REGION Network 69: EM Status Homed
   RUNG wire#powerrail
      Contact( "Unit1.Em4.ControlNodes".mainPnP.preOperationCheck.partNoDetect1 )
      wire#w1
      Contact( "Unit1.Em4.ControlNodes".alignTable.preOperationCheck.partNoDetect1 )
      wire#w2
      Contact( "Unit1.Em4.ControlNodes".ngPnP.preOperationCheck.partNoDetect )
      wire#w3
      I_Contact( #unitStatus.specialFunctions.dryRun )
      wire#w4
      Coil( "Unit1.Em4.ControlNodes".em.status.homed )
      Coil( #emFeedback.status.homed )
   END_RUNG
   RUNG wire#powerrail
      Contact( "Unit1.Em4.ControlNodes".mainPnP.preOperationCheck.partNoDetect2 )
   END_RUNG wire#w1
   RUNG wire#powerrail
      Contact( "Unit1.Em4.ControlNodes".mainPnP.preOperationCheck.partDetect1 )
   END_RUNG wire#w1
   RUNG wire#powerrail
      Contact( "Unit1.Em4.ControlNodes".mainPnP.preOperationCheck.partDetect2 )
   END_RUNG wire#w1
   RUNG wire#powerrail
      Contact( "Unit1.Em4.ControlNodes".mainPnP.preOperationCheck.partNG )
   END_RUNG wire#w1
   RUNG wire#powerrail
      Contact( "Unit1.Em4.ControlNodes".mainPnP.preOperationCheck.PartDetect1_1 )
   END_RUNG wire#w1
   RUNG wire#w1
      Contact( "Unit1.Em4.ControlNodes".alignTable.preOperationCheck.partDetect1 )
   END_RUNG wire#w2
   RUNG wire#w1
      Contact( "Unit1.Em4.ControlNodes".alignTable.preOperationCheck.partDetect2 )
   END_RUNG wire#w2
   RUNG wire#w2
      Contact( "Unit1.Em4.ControlNodes".ngPnP.preOperationCheck.partDetect )
   END_RUNG wire#w3
   RUNG wire#powerrail
      Contact( #unitStatus.specialFunctions.dryRun )
   END_RUNG wire#w4
   // the same network as SCL:
   "Unit1.Em4.ControlNodes".em.status.homed := (("Unit1.Em4.ControlNodes".mainPnP.preOperationCheck.partNoDetect1 OR "Unit1.Em4.ControlNodes".mainPnP.preOperationCheck.partNoDetect2 OR "Unit1.Em4.ControlNodes".mainPnP.preOperationCheck.partDetect1 OR "Unit1.Em4.ControlNodes".mainPnP.preOperationCheck.partDetect2 OR "Unit1.Em4.ControlNodes".mainPnP.preOperationCheck.partNG OR "Unit1.Em4.ControlNodes".mainPnP.preOperationCheck.PartDetect1_1) AND ("Unit1.Em4.ControlNodes".alignTable.preOperationCheck.partNoDetect1 OR "Unit1.Em4.ControlNodes".alignTable.preOperationCheck.partDetect1 OR "Unit1.Em4.ControlNodes".alignTable.preOperationCheck.partDetect2) AND ("Unit1.Em4.ControlNodes".ngPnP.preOperationCheck.partNoDetect OR "Unit1.Em4.ControlNodes".ngPnP.preOperationCheck.partDetect) AND NOT #unitStatus.specialFunctions.dryRun) OR #unitStatus.specialFunctions.dryRun;
   #emFeedback.status.homed := "Unit1.Em4.ControlNodes".em.status.homed;
END_REGION

REGION Network 70: EM Status Motion Ready
   RUNG wire#powerrail
      I_Contact( #instMainPnPHomeJob10.jobStatus.active )
      I_Contact( #instMainPnPLoadJob2.jobStatus.active )
      I_Contact( #instMainPnPUnloadJob3.jobStatus.active )
      I_Contact( #instMainPnPAvoidJob4.jobStatus.active )
      I_Contact( #instMainPnPOneLoadJob5.jobStatus.active )
      I_Contact( #instMainPnPOneUnLoadJob6.jobStatus.active )
      I_Contact( #instMainPnPDownWaitJob7.jobStatus.active )
      Coil( "Unit1.EmNodes".emRelations.em04."Bool"[10] )
   END_RUNG
   // the same network as SCL:
   "Unit1.EmNodes".emRelations.em04."Bool"[10] := NOT #instMainPnPHomeJob10.jobStatus.active AND NOT #instMainPnPLoadJob2.jobStatus.active AND NOT #instMainPnPUnloadJob3.jobStatus.active AND NOT #instMainPnPAvoidJob4.jobStatus.active AND NOT #instMainPnPOneLoadJob5.jobStatus.active AND NOT #instMainPnPOneUnLoadJob6.jobStatus.active AND NOT #instMainPnPDownWaitJob7.jobStatus.active;
END_REGION

REGION Network 72: Call Sequence [Main P&P]
   // Call the sequence. This contains the main logic of the equipment module
   RUNG wire#powerrail
      #InstSequenceMainPnP()
   END_RUNG
   // the same network as SCL:
   #InstSequenceMainPnP();   // "Unit1.Em4.Sequence_1_MainPnP"
END_REGION

REGION Network 73: Call Sequence [Align Table]
   // Call the sequence. This contains the main logic of the equipment module
   RUNG wire#powerrail
      #InstSequenceAlignTable()
   END_RUNG
   // the same network as SCL:
   #InstSequenceAlignTable();   // "Unit1.Em4.Sequence_2_AlignTable"
END_REGION

REGION Network 74: Call Sequence [NG P&P]
   // Call the sequence. This contains the main logic of the equipment module
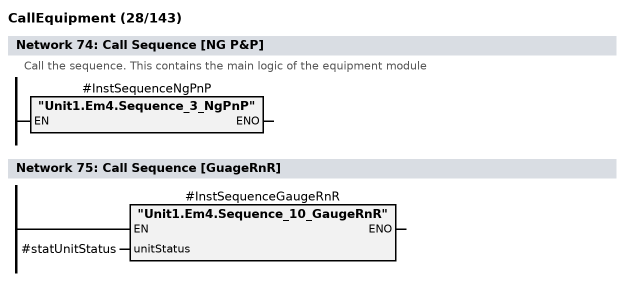
   RUNG wire#powerrail
      #InstSequenceNgPnP()
   END_RUNG
   // the same network as SCL:
   #InstSequenceNgPnP();   // "Unit1.Em4.Sequence_3_NgPnP"
END_REGION

REGION Network 75: Call Sequence [GuageRnR]
   RUNG wire#powerrail
      #InstSequenceGaugeRnR(unitStatus := #statUnitStatus)
   END_RUNG
   // the same network as SCL:
   #InstSequenceGaugeRnR(unitStatus := #statUnitStatus);   // "Unit1.Em4.Sequence_10_GaugeRnR"
END_REGION

REGION Network 76: *************** Control Modules (Axis) *******************
   // Call control modules that are actuators after the em logic (jobs and sequence), so that the latest commands are applied to the actuators.
END_REGION

REGION Network 77: Reset CMS
   // Reset Axis when the unit is in the resetting state.
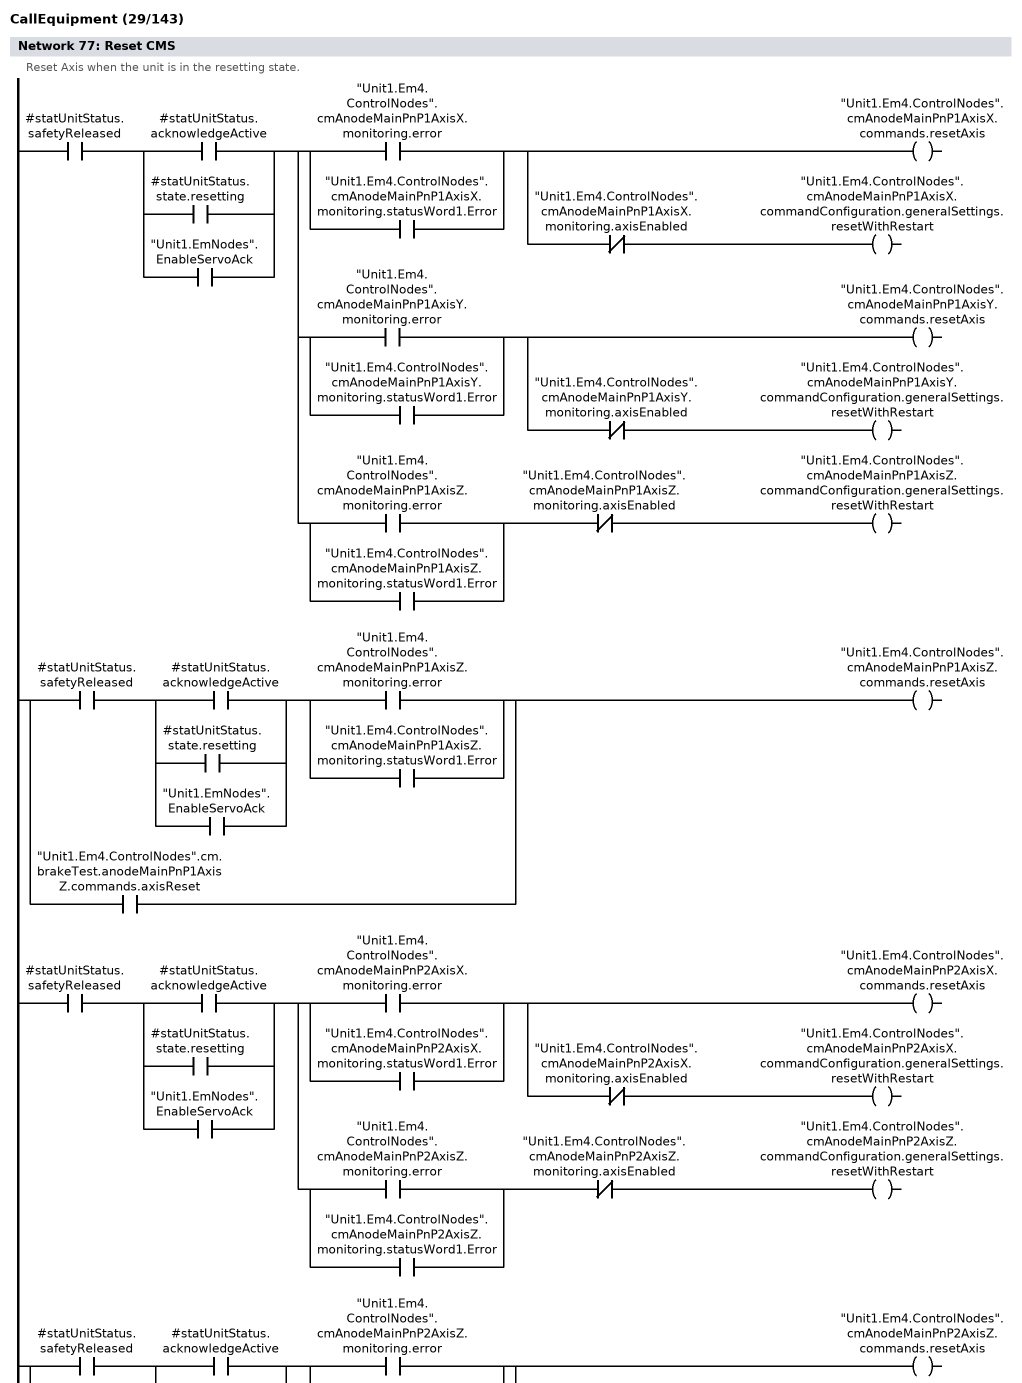
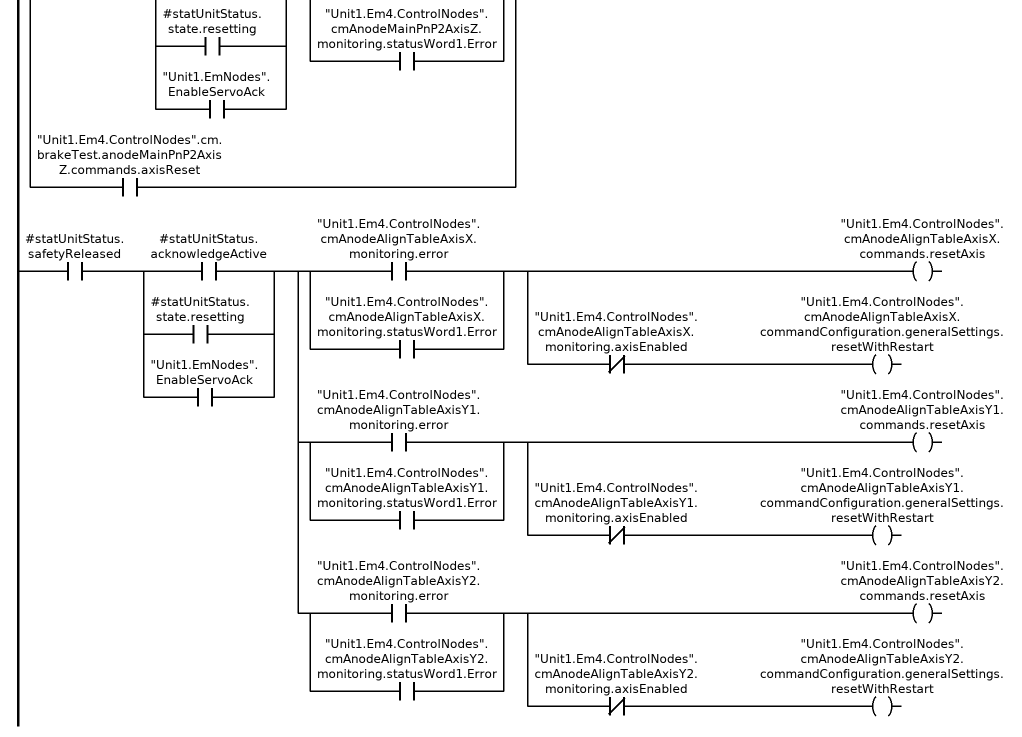
   RUNG wire#powerrail
      Contact( #statUnitStatus.safetyReleased )
      wire#w1
      Contact( #statUnitStatus.acknowledgeActive )
      wire#w2
      Contact( "Unit1.Em4.ControlNodes".cmAnodeMainPnP1AxisX.monitoring.error )
      wire#w3
      Coil( "Unit1.Em4.ControlNodes".cmAnodeMainPnP1AxisX.commands.resetAxis )
   END_RUNG
   RUNG wire#w1
      Contact( #statUnitStatus.state.resetting )
   END_RUNG wire#w2
   RUNG wire#w1
      Contact( "Unit1.EmNodes".EnableServoAck )
   END_RUNG wire#w2
   RUNG wire#w2
      Contact( "Unit1.Em4.ControlNodes".cmAnodeMainPnP1AxisX.monitoring.statusWord1.Error )
   END_RUNG wire#w3
   RUNG wire#w3
      I_Contact( "Unit1.Em4.ControlNodes".cmAnodeMainPnP1AxisX.monitoring.axisEnabled )
      Coil( "Unit1.Em4.ControlNodes".cmAnodeMainPnP1AxisX.commandConfiguration.generalSettings.resetWithRestart )
   END_RUNG
   RUNG wire#w2
      Contact( "Unit1.Em4.ControlNodes".cmAnodeMainPnP1AxisY.monitoring.error )
      wire#w4
      Coil( "Unit1.Em4.ControlNodes".cmAnodeMainPnP1AxisY.commands.resetAxis )
   END_RUNG
   RUNG wire#w2
      Contact( "Unit1.Em4.ControlNodes".cmAnodeMainPnP1AxisY.monitoring.statusWord1.Error )
   END_RUNG wire#w4
   RUNG wire#w4
      I_Contact( "Unit1.Em4.ControlNodes".cmAnodeMainPnP1AxisY.monitoring.axisEnabled )
      Coil( "Unit1.Em4.ControlNodes".cmAnodeMainPnP1AxisY.commandConfiguration.generalSettings.resetWithRestart )
   END_RUNG
   RUNG wire#w2
      Contact( "Unit1.Em4.ControlNodes".cmAnodeMainPnP1AxisZ.monitoring.error )
      wire#w5
      I_Contact( "Unit1.Em4.ControlNodes".cmAnodeMainPnP1AxisZ.monitoring.axisEnabled )
      Coil( "Unit1.Em4.ControlNodes".cmAnodeMainPnP1AxisZ.commandConfiguration.generalSettings.resetWithRestart )
   END_RUNG
   RUNG wire#w2
      Contact( "Unit1.Em4.ControlNodes".cmAnodeMainPnP1AxisZ.monitoring.statusWord1.Error )
   END_RUNG wire#w5
   RUNG wire#powerrail
      Contact( #statUnitStatus.safetyReleased )
      wire#w6
      Contact( #statUnitStatus.acknowledgeActive )
      wire#w7
      Contact( "Unit1.Em4.ControlNodes".cmAnodeMainPnP1AxisZ.monitoring.error )
      wire#w8
      Coil( "Unit1.Em4.ControlNodes".cmAnodeMainPnP1AxisZ.commands.resetAxis )
   END_RUNG
   RUNG wire#w6
      Contact( #statUnitStatus.state.resetting )
   END_RUNG wire#w7
   RUNG wire#w6
      Contact( "Unit1.EmNodes".EnableServoAck )
   END_RUNG wire#w7
   RUNG wire#w7
      Contact( "Unit1.Em4.ControlNodes".cmAnodeMainPnP1AxisZ.monitoring.statusWord1.Error )
   END_RUNG wire#w8
   RUNG wire#powerrail
      Contact( "Unit1.Em4.ControlNodes".cm.brakeTest.anodeMainPnP1AxisZ.commands.axisReset )
   END_RUNG wire#w8
   RUNG wire#powerrail
      Contact( #statUnitStatus.safetyReleased )
      wire#w9
      Contact( #statUnitStatus.acknowledgeActive )
      wire#w10
      Contact( "Unit1.Em4.ControlNodes".cmAnodeMainPnP2AxisX.monitoring.error )
      wire#w11
      Coil( "Unit1.Em4.ControlNodes".cmAnodeMainPnP2AxisX.commands.resetAxis )
   END_RUNG
   RUNG wire#w9
      Contact( #statUnitStatus.state.resetting )
   END_RUNG wire#w10
   RUNG wire#w9
      Contact( "Unit1.EmNodes".EnableServoAck )
   END_RUNG wire#w10
   RUNG wire#w10
      Contact( "Unit1.Em4.ControlNodes".cmAnodeMainPnP2AxisX.monitoring.statusWord1.Error )
   END_RUNG wire#w11
   RUNG wire#w11
      I_Contact( "Unit1.Em4.ControlNodes".cmAnodeMainPnP2AxisX.monitoring.axisEnabled )
      Coil( "Unit1.Em4.ControlNodes".cmAnodeMainPnP2AxisX.commandConfiguration.generalSettings.resetWithRestart )
   END_RUNG
   RUNG wire#w10
      Contact( "Unit1.Em4.ControlNodes".cmAnodeMainPnP2AxisZ.monitoring.error )
      wire#w12
      I_Contact( "Unit1.Em4.ControlNodes".cmAnodeMainPnP2AxisZ.monitoring.axisEnabled )
      Coil( "Unit1.Em4.ControlNodes".cmAnodeMainPnP2AxisZ.commandConfiguration.generalSettings.resetWithRestart )
   END_RUNG
   RUNG wire#w10
      Contact( "Unit1.Em4.ControlNodes".cmAnodeMainPnP2AxisZ.monitoring.statusWord1.Error )
   END_RUNG wire#w12
   RUNG wire#powerrail
      Contact( #statUnitStatus.safetyReleased )
      wire#w13
      Contact( #statUnitStatus.acknowledgeActive )
      wire#w14
      Contact( "Unit1.Em4.ControlNodes".cmAnodeMainPnP2AxisZ.monitoring.error )
      wire#w15
      Coil( "Unit1.Em4.ControlNodes".cmAnodeMainPnP2AxisZ.commands.resetAxis )
   END_RUNG
   RUNG wire#w13
      Contact( #statUnitStatus.state.resetting )
   END_RUNG wire#w14
   RUNG wire#w13
      Contact( "Unit1.EmNodes".EnableServoAck )
   END_RUNG wire#w14
   RUNG wire#w14
      Contact( "Unit1.Em4.ControlNodes".cmAnodeMainPnP2AxisZ.monitoring.statusWord1.Error )
   END_RUNG wire#w15
   RUNG wire#powerrail
      Contact( "Unit1.Em4.ControlNodes".cm.brakeTest.anodeMainPnP2AxisZ.commands.axisReset )
   END_RUNG wire#w15
   RUNG wire#powerrail
      Contact( #statUnitStatus.safetyReleased )
      wire#w16
      Contact( #statUnitStatus.acknowledgeActive )
      wire#w17
      Contact( "Unit1.Em4.ControlNodes".cmAnodeAlignTableAxisX.monitoring.error )
      wire#w18
      Coil( "Unit1.Em4.ControlNodes".cmAnodeAlignTableAxisX.commands.resetAxis )
   END_RUNG
   RUNG wire#w16
      Contact( #statUnitStatus.state.resetting )
   END_RUNG wire#w17
   RUNG wire#w16
      Contact( "Unit1.EmNodes".EnableServoAck )
   END_RUNG wire#w17
   RUNG wire#w17
      Contact( "Unit1.Em4.ControlNodes".cmAnodeAlignTableAxisX.monitoring.statusWord1.Error )
   END_RUNG wire#w18
   RUNG wire#w18
      I_Contact( "Unit1.Em4.ControlNodes".cmAnodeAlignTableAxisX.monitoring.axisEnabled )
      Coil( "Unit1.Em4.ControlNodes".cmAnodeAlignTableAxisX.commandConfiguration.generalSettings.resetWithRestart )
   END_RUNG
   RUNG wire#w17
      Contact( "Unit1.Em4.ControlNodes".cmAnodeAlignTableAxisY1.monitoring.error )
      wire#w19
      Coil( "Unit1.Em4.ControlNodes".cmAnodeAlignTableAxisY1.commands.resetAxis )
   END_RUNG
   RUNG wire#w17
      Contact( "Unit1.Em4.ControlNodes".cmAnodeAlignTableAxisY1.monitoring.statusWord1.Error )
   END_RUNG wire#w19
   RUNG wire#w19
      I_Contact( "Unit1.Em4.ControlNodes".cmAnodeAlignTableAxisY1.monitoring.axisEnabled )
      Coil( "Unit1.Em4.ControlNodes".cmAnodeAlignTableAxisY1.commandConfiguration.generalSettings.resetWithRestart )
   END_RUNG
   RUNG wire#w17
      Contact( "Unit1.Em4.ControlNodes".cmAnodeAlignTableAxisY2.monitoring.error )
      wire#w20
      Coil( "Unit1.Em4.ControlNodes".cmAnodeAlignTableAxisY2.commands.resetAxis )
   END_RUNG
   RUNG wire#w17
      Contact( "Unit1.Em4.ControlNodes".cmAnodeAlignTableAxisY2.monitoring.statusWord1.Error )
   END_RUNG wire#w20
   RUNG wire#w20
      I_Contact( "Unit1.Em4.ControlNodes".cmAnodeAlignTableAxisY2.monitoring.axisEnabled )
      Coil( "Unit1.Em4.ControlNodes".cmAnodeAlignTableAxisY2.commandConfiguration.generalSettings.resetWithRestart )
   END_RUNG
   // the same network as SCL:
   #_w1 := #statUnitStatus.safetyReleased AND (#statUnitStatus.acknowledgeActive OR #statUnitStatus.state.resetting OR "Unit1.EmNodes".EnableServoAck);
   "Unit1.Em4.ControlNodes".cmAnodeMainPnP1AxisX.commands.resetAxis := #_w1 AND ("Unit1.Em4.ControlNodes".cmAnodeMainPnP1AxisX.monitoring.error OR "Unit1.Em4.ControlNodes".cmAnodeMainPnP1AxisX.monitoring.statusWord1.Error);
   "Unit1.Em4.ControlNodes".cmAnodeMainPnP1AxisX.commandConfiguration.generalSettings.resetWithRestart := "Unit1.Em4.ControlNodes".cmAnodeMainPnP1AxisX.commands.resetAxis AND NOT "Unit1.Em4.ControlNodes".cmAnodeMainPnP1AxisX.monitoring.axisEnabled;
   "Unit1.Em4.ControlNodes".cmAnodeMainPnP1AxisY.commands.resetAxis := #_w1 AND ("Unit1.Em4.ControlNodes".cmAnodeMainPnP1AxisY.monitoring.error OR "Unit1.Em4.ControlNodes".cmAnodeMainPnP1AxisY.monitoring.statusWord1.Error);
   "Unit1.Em4.ControlNodes".cmAnodeMainPnP1AxisY.commandConfiguration.generalSettings.resetWithRestart := "Unit1.Em4.ControlNodes".cmAnodeMainPnP1AxisY.commands.resetAxis AND NOT "Unit1.Em4.ControlNodes".cmAnodeMainPnP1AxisY.monitoring.axisEnabled;
   "Unit1.Em4.ControlNodes".cmAnodeMainPnP1AxisZ.commandConfiguration.generalSettings.resetWithRestart := #_w1 AND ("Unit1.Em4.ControlNodes".cmAnodeMainPnP1AxisZ.monitoring.error OR "Unit1.Em4.ControlNodes".cmAnodeMainPnP1AxisZ.monitoring.statusWord1.Error) AND NOT "Unit1.Em4.ControlNodes".cmAnodeMainPnP1AxisZ.monitoring.axisEnabled;
   "Unit1.Em4.ControlNodes".cmAnodeMainPnP1AxisZ.commands.resetAxis := (#statUnitStatus.safetyReleased AND (#statUnitStatus.acknowledgeActive OR #statUnitStatus.state.resetting OR "Unit1.EmNodes".EnableServoAck) AND ("Unit1.Em4.ControlNodes".cmAnodeMainPnP1AxisZ.monitoring.error OR "Unit1.Em4.ControlNodes".cmAnodeMainPnP1AxisZ.monitoring.statusWord1.Error)) OR "Unit1.Em4.ControlNodes".cm.brakeTest.anodeMainPnP1AxisZ.commands.axisReset;
   #_w2 := #statUnitStatus.safetyReleased AND (#statUnitStatus.acknowledgeActive OR #statUnitStatus.state.resetting OR "Unit1.EmNodes".EnableServoAck);
   "Unit1.Em4.ControlNodes".cmAnodeMainPnP2AxisX.commands.resetAxis := #_w2 AND ("Unit1.Em4.ControlNodes".cmAnodeMainPnP2AxisX.monitoring.error OR "Unit1.Em4.ControlNodes".cmAnodeMainPnP2AxisX.monitoring.statusWord1.Error);
   "Unit1.Em4.ControlNodes".cmAnodeMainPnP2AxisX.commandConfiguration.generalSettings.resetWithRestart := "Unit1.Em4.ControlNodes".cmAnodeMainPnP2AxisX.commands.resetAxis AND NOT "Unit1.Em4.ControlNodes".cmAnodeMainPnP2AxisX.monitoring.axisEnabled;
   "Unit1.Em4.ControlNodes".cmAnodeMainPnP2AxisZ.commandConfiguration.generalSettings.resetWithRestart := #_w2 AND ("Unit1.Em4.ControlNodes".cmAnodeMainPnP2AxisZ.monitoring.error OR "Unit1.Em4.ControlNodes".cmAnodeMainPnP2AxisZ.monitoring.statusWord1.Error) AND NOT "Unit1.Em4.ControlNodes".cmAnodeMainPnP2AxisZ.monitoring.axisEnabled;
   "Unit1.Em4.ControlNodes".cmAnodeMainPnP2AxisZ.commands.resetAxis := (#statUnitStatus.safetyReleased AND (#statUnitStatus.acknowledgeActive OR #statUnitStatus.state.resetting OR "Unit1.EmNodes".EnableServoAck) AND ("Unit1.Em4.ControlNodes".cmAnodeMainPnP2AxisZ.monitoring.error OR "Unit1.Em4.ControlNodes".cmAnodeMainPnP2AxisZ.monitoring.statusWord1.Error)) OR "Unit1.Em4.ControlNodes".cm.brakeTest.anodeMainPnP2AxisZ.commands.axisReset;
   #_w3 := #statUnitStatus.safetyReleased AND (#statUnitStatus.acknowledgeActive OR #statUnitStatus.state.resetting OR "Unit1.EmNodes".EnableServoAck);
   "Unit1.Em4.ControlNodes".cmAnodeAlignTableAxisX.commands.resetAxis := #_w3 AND ("Unit1.Em4.ControlNodes".cmAnodeAlignTableAxisX.monitoring.error OR "Unit1.Em4.ControlNodes".cmAnodeAlignTableAxisX.monitoring.statusWord1.Error);
   "Unit1.Em4.ControlNodes".cmAnodeAlignTableAxisX.commandConfiguration.generalSettings.resetWithRestart := "Unit1.Em4.ControlNodes".cmAnodeAlignTableAxisX.commands.resetAxis AND NOT "Unit1.Em4.ControlNodes".cmAnodeAlignTableAxisX.monitoring.axisEnabled;
   "Unit1.Em4.ControlNodes".cmAnodeAlignTableAxisY1.commands.resetAxis := #_w3 AND ("Unit1.Em4.ControlNodes".cmAnodeAlignTableAxisY1.monitoring.error OR "Unit1.Em4.ControlNodes".cmAnodeAlignTableAxisY1.monitoring.statusWord1.Error);
   "Unit1.Em4.ControlNodes".cmAnodeAlignTableAxisY1.commandConfiguration.generalSettings.resetWithRestart := "Unit1.Em4.ControlNodes".cmAnodeAlignTableAxisY1.commands.resetAxis AND NOT "Unit1.Em4.ControlNodes".cmAnodeAlignTableAxisY1.monitoring.axisEnabled;
   "Unit1.Em4.ControlNodes".cmAnodeAlignTableAxisY2.commands.resetAxis := #_w3 AND ("Unit1.Em4.ControlNodes".cmAnodeAlignTableAxisY2.monitoring.error OR "Unit1.Em4.ControlNodes".cmAnodeAlignTableAxisY2.monitoring.statusWord1.Error);
   "Unit1.Em4.ControlNodes".cmAnodeAlignTableAxisY2.commandConfiguration.generalSettings.resetWithRestart := "Unit1.Em4.ControlNodes".cmAnodeAlignTableAxisY2.commands.resetAxis AND NOT "Unit1.Em4.ControlNodes".cmAnodeAlignTableAxisY2.monitoring.axisEnabled;
END_REGION

REGION Network 78: Enable/Disable CMs
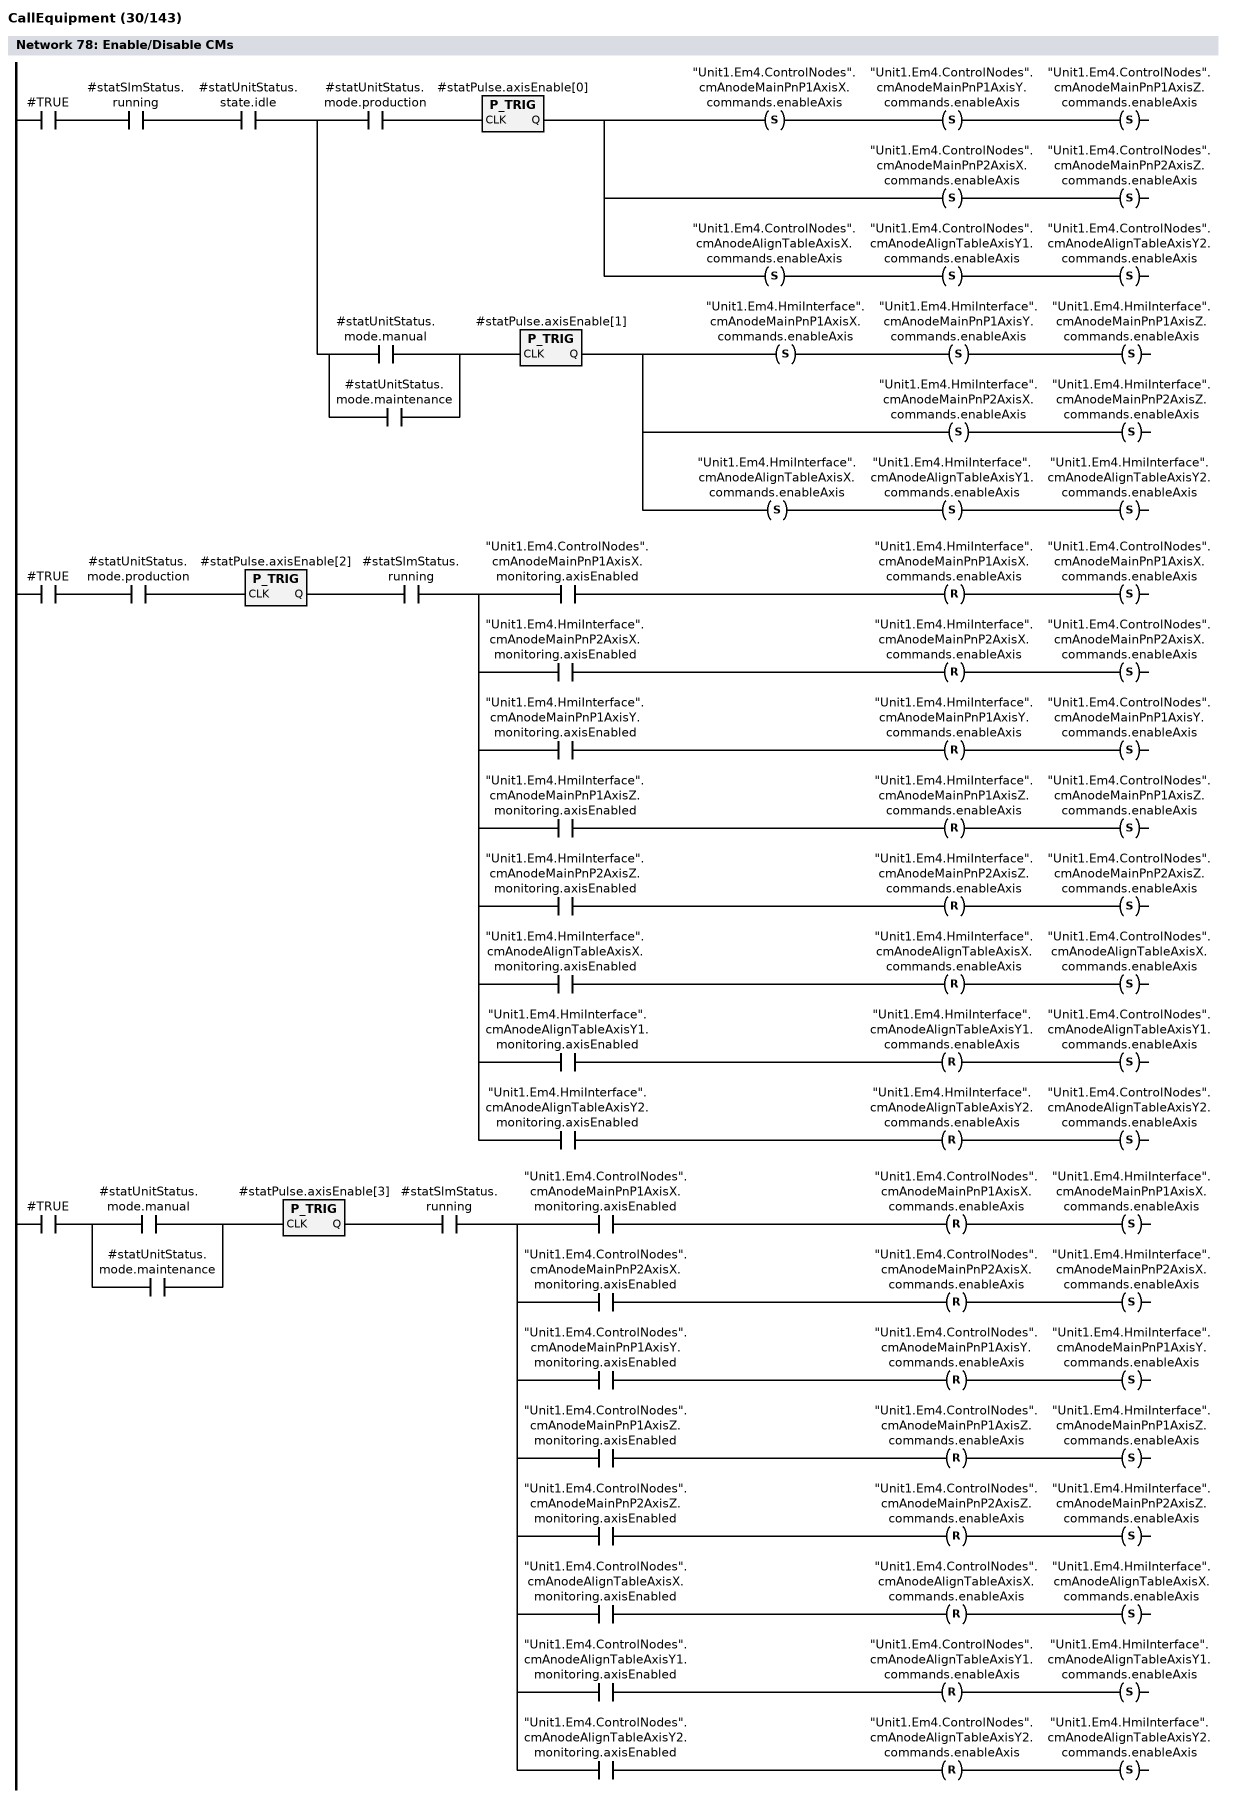
   RUNG wire#powerrail
      Contact( #TRUE )
      Contact( #statSlmStatus.running )
      Contact( #statUnitStatus.state.idle )
      wire#w1
      Contact( #statUnitStatus.mode.production )
      P_Trig( #statPulse.axisEnable[0] )
      wire#w2
      S_Coil( "Unit1.Em4.ControlNodes".cmAnodeMainPnP1AxisX.commands.enableAxis )
      S_Coil( "Unit1.Em4.ControlNodes".cmAnodeMainPnP1AxisY.commands.enableAxis )
      S_Coil( "Unit1.Em4.ControlNodes".cmAnodeMainPnP1AxisZ.commands.enableAxis )
   END_RUNG
   RUNG wire#w2
      S_Coil( "Unit1.Em4.ControlNodes".cmAnodeMainPnP2AxisX.commands.enableAxis )
      S_Coil( "Unit1.Em4.ControlNodes".cmAnodeMainPnP2AxisZ.commands.enableAxis )
   END_RUNG
   RUNG wire#w2
      S_Coil( "Unit1.Em4.ControlNodes".cmAnodeAlignTableAxisX.commands.enableAxis )
      S_Coil( "Unit1.Em4.ControlNodes".cmAnodeAlignTableAxisY1.commands.enableAxis )
      S_Coil( "Unit1.Em4.ControlNodes".cmAnodeAlignTableAxisY2.commands.enableAxis )
   END_RUNG
   RUNG wire#w1
      Contact( #statUnitStatus.mode.manual )
      wire#w3
      P_Trig( #statPulse.axisEnable[1] )
      wire#w4
      S_Coil( "Unit1.Em4.HmiInterface".cmAnodeMainPnP1AxisX.commands.enableAxis )
      S_Coil( "Unit1.Em4.HmiInterface".cmAnodeMainPnP1AxisY.commands.enableAxis )
      S_Coil( "Unit1.Em4.HmiInterface".cmAnodeMainPnP1AxisZ.commands.enableAxis )
   END_RUNG
   RUNG wire#w1
      Contact( #statUnitStatus.mode.maintenance )
   END_RUNG wire#w3
   RUNG wire#w4
      S_Coil( "Unit1.Em4.HmiInterface".cmAnodeMainPnP2AxisX.commands.enableAxis )
      S_Coil( "Unit1.Em4.HmiInterface".cmAnodeMainPnP2AxisZ.commands.enableAxis )
   END_RUNG
   RUNG wire#w4
      S_Coil( "Unit1.Em4.HmiInterface".cmAnodeAlignTableAxisX.commands.enableAxis )
      S_Coil( "Unit1.Em4.HmiInterface".cmAnodeAlignTableAxisY1.commands.enableAxis )
      S_Coil( "Unit1.Em4.HmiInterface".cmAnodeAlignTableAxisY2.commands.enableAxis )
   END_RUNG
   RUNG wire#powerrail
      Contact( #TRUE )
      Contact( #statUnitStatus.mode.production )
      P_Trig( #statPulse.axisEnable[2] )
      Contact( #statSlmStatus.running )
      wire#w5
      Contact( "Unit1.Em4.ControlNodes".cmAnodeMainPnP1AxisX.monitoring.axisEnabled )
      R_Coil( "Unit1.Em4.HmiInterface".cmAnodeMainPnP1AxisX.commands.enableAxis )
      S_Coil( "Unit1.Em4.ControlNodes".cmAnodeMainPnP1AxisX.commands.enableAxis )
   END_RUNG
   RUNG wire#w5
      Contact( "Unit1.Em4.HmiInterface".cmAnodeMainPnP2AxisX.monitoring.axisEnabled )
      R_Coil( "Unit1.Em4.HmiInterface".cmAnodeMainPnP2AxisX.commands.enableAxis )
      S_Coil( "Unit1.Em4.ControlNodes".cmAnodeMainPnP2AxisX.commands.enableAxis )
   END_RUNG
   RUNG wire#w5
      Contact( "Unit1.Em4.HmiInterface".cmAnodeMainPnP1AxisY.monitoring.axisEnabled )
      R_Coil( "Unit1.Em4.HmiInterface".cmAnodeMainPnP1AxisY.commands.enableAxis )
      S_Coil( "Unit1.Em4.ControlNodes".cmAnodeMainPnP1AxisY.commands.enableAxis )
   END_RUNG
   RUNG wire#w5
      Contact( "Unit1.Em4.HmiInterface".cmAnodeMainPnP1AxisZ.monitoring.axisEnabled )
      R_Coil( "Unit1.Em4.HmiInterface".cmAnodeMainPnP1AxisZ.commands.enableAxis )
      S_Coil( "Unit1.Em4.ControlNodes".cmAnodeMainPnP1AxisZ.commands.enableAxis )
   END_RUNG
   RUNG wire#w5
      Contact( "Unit1.Em4.HmiInterface".cmAnodeMainPnP2AxisZ.monitoring.axisEnabled )
      R_Coil( "Unit1.Em4.HmiInterface".cmAnodeMainPnP2AxisZ.commands.enableAxis )
      S_Coil( "Unit1.Em4.ControlNodes".cmAnodeMainPnP2AxisZ.commands.enableAxis )
   END_RUNG
   RUNG wire#w5
      Contact( "Unit1.Em4.HmiInterface".cmAnodeAlignTableAxisX.monitoring.axisEnabled )
      R_Coil( "Unit1.Em4.HmiInterface".cmAnodeAlignTableAxisX.commands.enableAxis )
      S_Coil( "Unit1.Em4.ControlNodes".cmAnodeAlignTableAxisX.commands.enableAxis )
   END_RUNG
   RUNG wire#w5
      Contact( "Unit1.Em4.HmiInterface".cmAnodeAlignTableAxisY1.monitoring.axisEnabled )
      R_Coil( "Unit1.Em4.HmiInterface".cmAnodeAlignTableAxisY1.commands.enableAxis )
      S_Coil( "Unit1.Em4.ControlNodes".cmAnodeAlignTableAxisY1.commands.enableAxis )
   END_RUNG
   RUNG wire#w5
      Contact( "Unit1.Em4.HmiInterface".cmAnodeAlignTableAxisY2.monitoring.axisEnabled )
      R_Coil( "Unit1.Em4.HmiInterface".cmAnodeAlignTableAxisY2.commands.enableAxis )
      S_Coil( "Unit1.Em4.ControlNodes".cmAnodeAlignTableAxisY2.commands.enableAxis )
   END_RUNG
   RUNG wire#powerrail
      Contact( #TRUE )
      wire#w6
      Contact( #statUnitStatus.mode.manual )
      wire#w7
      P_Trig( #statPulse.axisEnable[3] )
      Contact( #statSlmStatus.running )
      wire#w8
      Contact( "Unit1.Em4.ControlNodes".cmAnodeMainPnP1AxisX.monitoring.axisEnabled )
      R_Coil( "Unit1.Em4.ControlNodes".cmAnodeMainPnP1AxisX.commands.enableAxis )
      S_Coil( "Unit1.Em4.HmiInterface".cmAnodeMainPnP1AxisX.commands.enableAxis )
   END_RUNG
   RUNG wire#w6
      Contact( #statUnitStatus.mode.maintenance )
   END_RUNG wire#w7
   RUNG wire#w8
      Contact( "Unit1.Em4.ControlNodes".cmAnodeMainPnP2AxisX.monitoring.axisEnabled )
      R_Coil( "Unit1.Em4.ControlNodes".cmAnodeMainPnP2AxisX.commands.enableAxis )
      S_Coil( "Unit1.Em4.HmiInterface".cmAnodeMainPnP2AxisX.commands.enableAxis )
   END_RUNG
   RUNG wire#w8
      Contact( "Unit1.Em4.ControlNodes".cmAnodeMainPnP1AxisY.monitoring.axisEnabled )
      R_Coil( "Unit1.Em4.ControlNodes".cmAnodeMainPnP1AxisY.commands.enableAxis )
      S_Coil( "Unit1.Em4.HmiInterface".cmAnodeMainPnP1AxisY.commands.enableAxis )
   END_RUNG
   RUNG wire#w8
      Contact( "Unit1.Em4.ControlNodes".cmAnodeMainPnP1AxisZ.monitoring.axisEnabled )
      R_Coil( "Unit1.Em4.ControlNodes".cmAnodeMainPnP1AxisZ.commands.enableAxis )
      S_Coil( "Unit1.Em4.HmiInterface".cmAnodeMainPnP1AxisZ.commands.enableAxis )
   END_RUNG
   RUNG wire#w8
      Contact( "Unit1.Em4.ControlNodes".cmAnodeMainPnP2AxisZ.monitoring.axisEnabled )
      R_Coil( "Unit1.Em4.ControlNodes".cmAnodeMainPnP2AxisZ.commands.enableAxis )
      S_Coil( "Unit1.Em4.HmiInterface".cmAnodeMainPnP2AxisZ.commands.enableAxis )
   END_RUNG
   RUNG wire#w8
      Contact( "Unit1.Em4.ControlNodes".cmAnodeAlignTableAxisX.monitoring.axisEnabled )
      R_Coil( "Unit1.Em4.ControlNodes".cmAnodeAlignTableAxisX.commands.enableAxis )
      S_Coil( "Unit1.Em4.HmiInterface".cmAnodeAlignTableAxisX.commands.enableAxis )
   END_RUNG
   RUNG wire#w8
      Contact( "Unit1.Em4.ControlNodes".cmAnodeAlignTableAxisY1.monitoring.axisEnabled )
      R_Coil( "Unit1.Em4.ControlNodes".cmAnodeAlignTableAxisY1.commands.enableAxis )
      S_Coil( "Unit1.Em4.HmiInterface".cmAnodeAlignTableAxisY1.commands.enableAxis )
   END_RUNG
   RUNG wire#w8
      Contact( "Unit1.Em4.ControlNodes".cmAnodeAlignTableAxisY2.monitoring.axisEnabled )
      R_Coil( "Unit1.Em4.ControlNodes".cmAnodeAlignTableAxisY2.commands.enableAxis )
      S_Coil( "Unit1.Em4.HmiInterface".cmAnodeAlignTableAxisY2.commands.enableAxis )
   END_RUNG
   // the same network as SCL:
   #_w1 := #TRUE AND #statSlmStatus.running AND #statUnitStatus.state.idle;
   #_w2 := #_w1 AND #statUnitStatus.mode.production;
   #_w3 := #_w2 AND NOT #statPulse.axisEnable[0];   // rising edge
   #statPulse.axisEnable[0] := #_w2;
   IF #_w3 THEN
       "Unit1.Em4.ControlNodes".cmAnodeMainPnP1AxisX.commands.enableAxis := TRUE;
       "Unit1.Em4.ControlNodes".cmAnodeMainPnP1AxisY.commands.enableAxis := TRUE;
       "Unit1.Em4.ControlNodes".cmAnodeMainPnP1AxisZ.commands.enableAxis := TRUE;
       "Unit1.Em4.ControlNodes".cmAnodeMainPnP2AxisX.commands.enableAxis := TRUE;
       "Unit1.Em4.ControlNodes".cmAnodeMainPnP2AxisZ.commands.enableAxis := TRUE;
       "Unit1.Em4.ControlNodes".cmAnodeAlignTableAxisX.commands.enableAxis := TRUE;
       "Unit1.Em4.ControlNodes".cmAnodeAlignTableAxisY1.commands.enableAxis := TRUE;
       "Unit1.Em4.ControlNodes".cmAnodeAlignTableAxisY2.commands.enableAxis := TRUE;
   END_IF;
   #_w4 := #_w1 AND (#statUnitStatus.mode.manual OR #statUnitStatus.mode.maintenance);
   #_w5 := #_w4 AND NOT #statPulse.axisEnable[1];   // rising edge
   #statPulse.axisEnable[1] := #_w4;
   IF #_w5 THEN
       "Unit1.Em4.HmiInterface".cmAnodeMainPnP1AxisX.commands.enableAxis := TRUE;
       "Unit1.Em4.HmiInterface".cmAnodeMainPnP1AxisY.commands.enableAxis := TRUE;
       "Unit1.Em4.HmiInterface".cmAnodeMainPnP1AxisZ.commands.enableAxis := TRUE;
       "Unit1.Em4.HmiInterface".cmAnodeMainPnP2AxisX.commands.enableAxis := TRUE;
       "Unit1.Em4.HmiInterface".cmAnodeMainPnP2AxisZ.commands.enableAxis := TRUE;
       "Unit1.Em4.HmiInterface".cmAnodeAlignTableAxisX.commands.enableAxis := TRUE;
       "Unit1.Em4.HmiInterface".cmAnodeAlignTableAxisY1.commands.enableAxis := TRUE;
       "Unit1.Em4.HmiInterface".cmAnodeAlignTableAxisY2.commands.enableAxis := TRUE;
   END_IF;
   #_w6 := #TRUE AND #statUnitStatus.mode.production;
   #_w7 := #_w6 AND NOT #statPulse.axisEnable[2];   // rising edge
   #statPulse.axisEnable[2] := #_w6;
   #_w8 := #_w7 AND #statSlmStatus.running;
   IF #_w8 AND "Unit1.Em4.ControlNodes".cmAnodeMainPnP1AxisX.monitoring.axisEnabled THEN
       "Unit1.Em4.HmiInterface".cmAnodeMainPnP1AxisX.commands.enableAxis := FALSE;
       "Unit1.Em4.ControlNodes".cmAnodeMainPnP1AxisX.commands.enableAxis := TRUE;
   END_IF;
   IF #_w8 AND "Unit1.Em4.HmiInterface".cmAnodeMainPnP2AxisX.monitoring.axisEnabled THEN
       "Unit1.Em4.HmiInterface".cmAnodeMainPnP2AxisX.commands.enableAxis := FALSE;
       "Unit1.Em4.ControlNodes".cmAnodeMainPnP2AxisX.commands.enableAxis := TRUE;
   END_IF;
   IF #_w8 AND "Unit1.Em4.HmiInterface".cmAnodeMainPnP1AxisY.monitoring.axisEnabled THEN
       "Unit1.Em4.HmiInterface".cmAnodeMainPnP1AxisY.commands.enableAxis := FALSE;
       "Unit1.Em4.ControlNodes".cmAnodeMainPnP1AxisY.commands.enableAxis := TRUE;
   END_IF;
   IF #_w8 AND "Unit1.Em4.HmiInterface".cmAnodeMainPnP1AxisZ.monitoring.axisEnabled THEN
       "Unit1.Em4.HmiInterface".cmAnodeMainPnP1AxisZ.commands.enableAxis := FALSE;
       "Unit1.Em4.ControlNodes".cmAnodeMainPnP1AxisZ.commands.enableAxis := TRUE;
   END_IF;
   IF #_w8 AND "Unit1.Em4.HmiInterface".cmAnodeMainPnP2AxisZ.monitoring.axisEnabled THEN
       "Unit1.Em4.HmiInterface".cmAnodeMainPnP2AxisZ.commands.enableAxis := FALSE;
       "Unit1.Em4.ControlNodes".cmAnodeMainPnP2AxisZ.commands.enableAxis := TRUE;
   END_IF;
   IF #_w8 AND "Unit1.Em4.HmiInterface".cmAnodeAlignTableAxisX.monitoring.axisEnabled THEN
       "Unit1.Em4.HmiInterface".cmAnodeAlignTableAxisX.commands.enableAxis := FALSE;
       "Unit1.Em4.ControlNodes".cmAnodeAlignTableAxisX.commands.enableAxis := TRUE;
   END_IF;
   IF #_w8 AND "Unit1.Em4.HmiInterface".cmAnodeAlignTableAxisY1.monitoring.axisEnabled THEN
       "Unit1.Em4.HmiInterface".cmAnodeAlignTableAxisY1.commands.enableAxis := FALSE;
       "Unit1.Em4.ControlNodes".cmAnodeAlignTableAxisY1.commands.enableAxis := TRUE;
   END_IF;
   IF #_w8 AND "Unit1.Em4.HmiInterface".cmAnodeAlignTableAxisY2.monitoring.axisEnabled THEN
       "Unit1.Em4.HmiInterface".cmAnodeAlignTableAxisY2.commands.enableAxis := FALSE;
       "Unit1.Em4.ControlNodes".cmAnodeAlignTableAxisY2.commands.enableAxis := TRUE;
   END_IF;
   #_w9 := #TRUE AND (#statUnitStatus.mode.manual OR #statUnitStatus.mode.maintenance);
   #_w10 := #_w9 AND NOT #statPulse.axisEnable[3];   // rising edge
   #statPulse.axisEnable[3] := #_w9;
   #_w11 := #_w10 AND #statSlmStatus.running;
   IF #_w11 AND "Unit1.Em4.ControlNodes".cmAnodeMainPnP1AxisX.monitoring.axisEnabled THEN
       "Unit1.Em4.ControlNodes".cmAnodeMainPnP1AxisX.commands.enableAxis := FALSE;
       "Unit1.Em4.HmiInterface".cmAnodeMainPnP1AxisX.commands.enableAxis := TRUE;
   END_IF;
   IF #_w11 AND "Unit1.Em4.ControlNodes".cmAnodeMainPnP2AxisX.monitoring.axisEnabled THEN
       "Unit1.Em4.ControlNodes".cmAnodeMainPnP2AxisX.commands.enableAxis := FALSE;
       "Unit1.Em4.HmiInterface".cmAnodeMainPnP2AxisX.commands.enableAxis := TRUE;
   END_IF;
   IF #_w11 AND "Unit1.Em4.ControlNodes".cmAnodeMainPnP1AxisY.monitoring.axisEnabled THEN
       "Unit1.Em4.ControlNodes".cmAnodeMainPnP1AxisY.commands.enableAxis := FALSE;
       "Unit1.Em4.HmiInterface".cmAnodeMainPnP1AxisY.commands.enableAxis := TRUE;
   END_IF;
   IF #_w11 AND "Unit1.Em4.ControlNodes".cmAnodeMainPnP1AxisZ.monitoring.axisEnabled THEN
       "Unit1.Em4.ControlNodes".cmAnodeMainPnP1AxisZ.commands.enableAxis := FALSE;
       "Unit1.Em4.HmiInterface".cmAnodeMainPnP1AxisZ.commands.enableAxis := TRUE;
   END_IF;
   IF #_w11 AND "Unit1.Em4.ControlNodes".cmAnodeMainPnP2AxisZ.monitoring.axisEnabled THEN
       "Unit1.Em4.ControlNodes".cmAnodeMainPnP2AxisZ.commands.enableAxis := FALSE;
       "Unit1.Em4.HmiInterface".cmAnodeMainPnP2AxisZ.commands.enableAxis := TRUE;
   END_IF;
   IF #_w11 AND "Unit1.Em4.ControlNodes".cmAnodeAlignTableAxisX.monitoring.axisEnabled THEN
       "Unit1.Em4.ControlNodes".cmAnodeAlignTableAxisX.commands.enableAxis := FALSE;
       "Unit1.Em4.HmiInterface".cmAnodeAlignTableAxisX.commands.enableAxis := TRUE;
   END_IF;
   IF #_w11 AND "Unit1.Em4.ControlNodes".cmAnodeAlignTableAxisY1.monitoring.axisEnabled THEN
       "Unit1.Em4.ControlNodes".cmAnodeAlignTableAxisY1.commands.enableAxis := FALSE;
       "Unit1.Em4.HmiInterface".cmAnodeAlignTableAxisY1.commands.enableAxis := TRUE;
   END_IF;
   IF #_w11 AND "Unit1.Em4.ControlNodes".cmAnodeAlignTableAxisY2.monitoring.axisEnabled THEN
       "Unit1.Em4.ControlNodes".cmAnodeAlignTableAxisY2.commands.enableAxis := FALSE;
       "Unit1.Em4.HmiInterface".cmAnodeAlignTableAxisY2.commands.enableAxis := TRUE;
   END_IF;
END_REGION

REGION Network 79: PHMI Servo Enable CMs
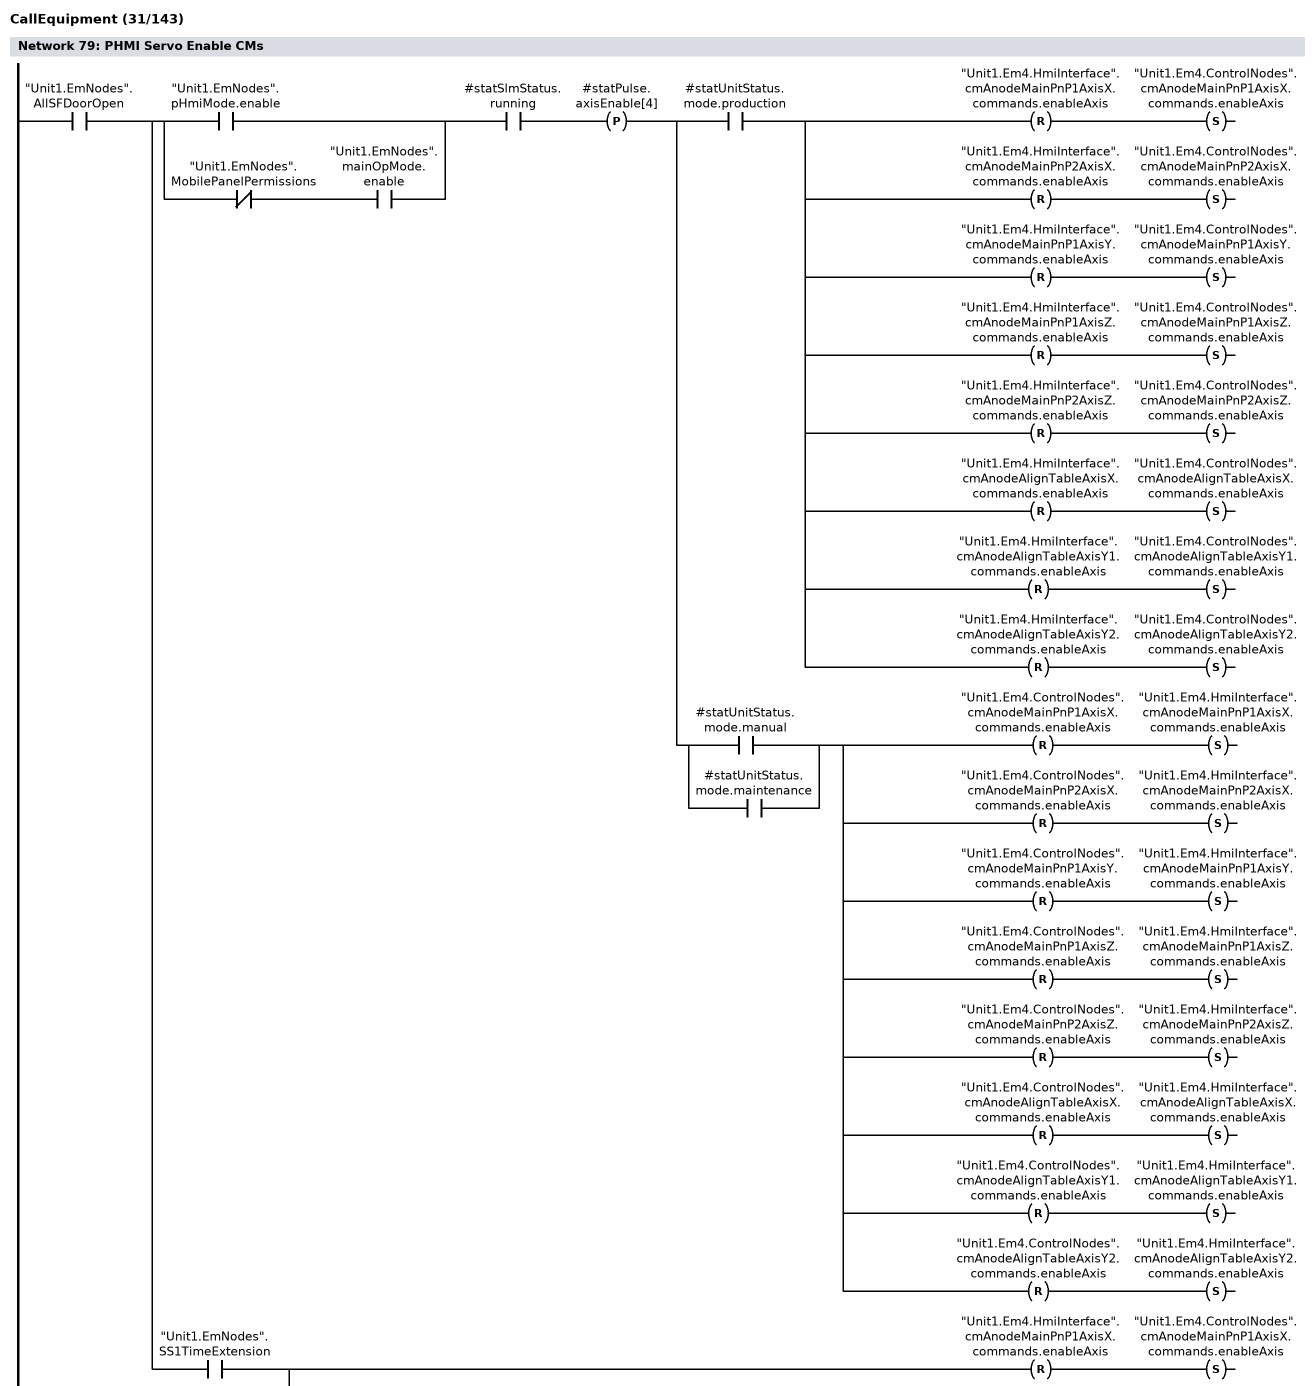
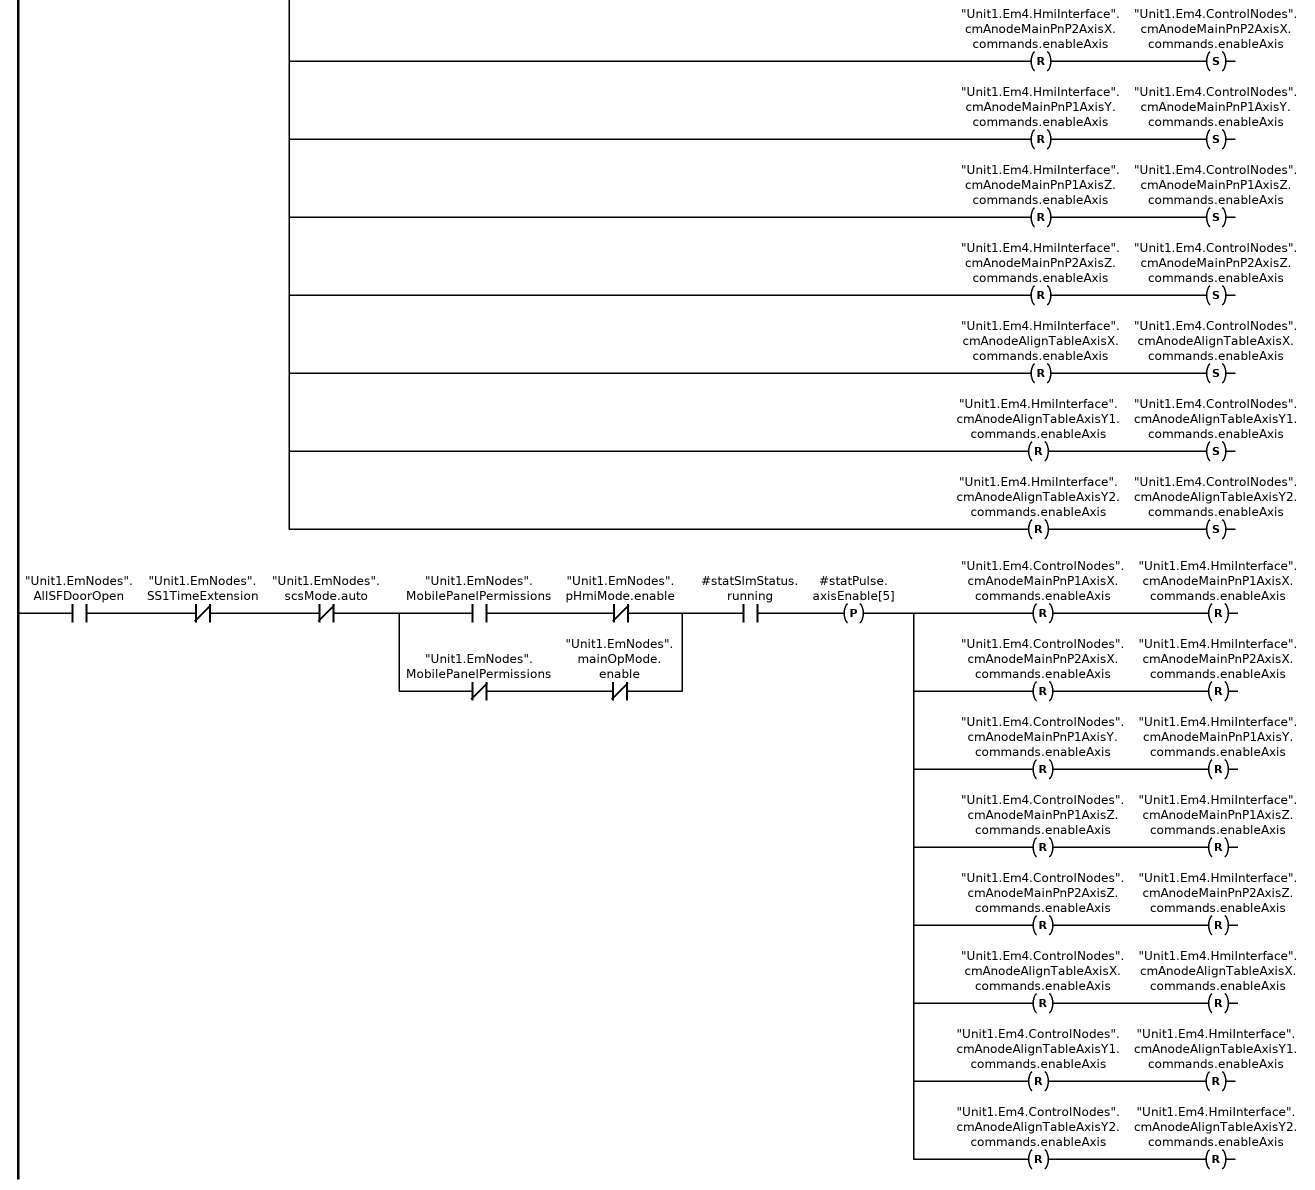
   RUNG wire#powerrail
      Contact( "Unit1.EmNodes".AllSFDoorOpen )
      wire#w1
      Contact( "Unit1.EmNodes".pHmiMode.enable )
      wire#w2
      Contact( #statSlmStatus.running )
      P_Trig( #statPulse.axisEnable[4] )
      wire#w3
      Contact( #statUnitStatus.mode.production )
      wire#w4
      R_Coil( "Unit1.Em4.HmiInterface".cmAnodeMainPnP1AxisX.commands.enableAxis )
      S_Coil( "Unit1.Em4.ControlNodes".cmAnodeMainPnP1AxisX.commands.enableAxis )
   END_RUNG
   RUNG wire#w1
      I_Contact( "Unit1.EmNodes".MobilePanelPermissions )
      Contact( "Unit1.EmNodes".mainOpMode.enable )
   END_RUNG wire#w2
   RUNG wire#w4
      R_Coil( "Unit1.Em4.HmiInterface".cmAnodeMainPnP2AxisX.commands.enableAxis )
      S_Coil( "Unit1.Em4.ControlNodes".cmAnodeMainPnP2AxisX.commands.enableAxis )
   END_RUNG
   RUNG wire#w4
      R_Coil( "Unit1.Em4.HmiInterface".cmAnodeMainPnP1AxisY.commands.enableAxis )
      S_Coil( "Unit1.Em4.ControlNodes".cmAnodeMainPnP1AxisY.commands.enableAxis )
   END_RUNG
   RUNG wire#w4
      R_Coil( "Unit1.Em4.HmiInterface".cmAnodeMainPnP1AxisZ.commands.enableAxis )
      S_Coil( "Unit1.Em4.ControlNodes".cmAnodeMainPnP1AxisZ.commands.enableAxis )
   END_RUNG
   RUNG wire#w4
      R_Coil( "Unit1.Em4.HmiInterface".cmAnodeMainPnP2AxisZ.commands.enableAxis )
      S_Coil( "Unit1.Em4.ControlNodes".cmAnodeMainPnP2AxisZ.commands.enableAxis )
   END_RUNG
   RUNG wire#w4
      R_Coil( "Unit1.Em4.HmiInterface".cmAnodeAlignTableAxisX.commands.enableAxis )
      S_Coil( "Unit1.Em4.ControlNodes".cmAnodeAlignTableAxisX.commands.enableAxis )
   END_RUNG
   RUNG wire#w4
      R_Coil( "Unit1.Em4.HmiInterface".cmAnodeAlignTableAxisY1.commands.enableAxis )
      S_Coil( "Unit1.Em4.ControlNodes".cmAnodeAlignTableAxisY1.commands.enableAxis )
   END_RUNG
   RUNG wire#w4
      R_Coil( "Unit1.Em4.HmiInterface".cmAnodeAlignTableAxisY2.commands.enableAxis )
      S_Coil( "Unit1.Em4.ControlNodes".cmAnodeAlignTableAxisY2.commands.enableAxis )
   END_RUNG
   RUNG wire#w3
      Contact( #statUnitStatus.mode.manual )
      wire#w5
      R_Coil( "Unit1.Em4.ControlNodes".cmAnodeMainPnP1AxisX.commands.enableAxis )
      S_Coil( "Unit1.Em4.HmiInterface".cmAnodeMainPnP1AxisX.commands.enableAxis )
   END_RUNG
   RUNG wire#w3
      Contact( #statUnitStatus.mode.maintenance )
   END_RUNG wire#w5
   RUNG wire#w5
      R_Coil( "Unit1.Em4.ControlNodes".cmAnodeMainPnP2AxisX.commands.enableAxis )
      S_Coil( "Unit1.Em4.HmiInterface".cmAnodeMainPnP2AxisX.commands.enableAxis )
   END_RUNG
   RUNG wire#w5
      R_Coil( "Unit1.Em4.ControlNodes".cmAnodeMainPnP1AxisY.commands.enableAxis )
      S_Coil( "Unit1.Em4.HmiInterface".cmAnodeMainPnP1AxisY.commands.enableAxis )
   END_RUNG
   RUNG wire#w5
      R_Coil( "Unit1.Em4.ControlNodes".cmAnodeMainPnP1AxisZ.commands.enableAxis )
      S_Coil( "Unit1.Em4.HmiInterface".cmAnodeMainPnP1AxisZ.commands.enableAxis )
   END_RUNG
   RUNG wire#w5
      R_Coil( "Unit1.Em4.ControlNodes".cmAnodeMainPnP2AxisZ.commands.enableAxis )
      S_Coil( "Unit1.Em4.HmiInterface".cmAnodeMainPnP2AxisZ.commands.enableAxis )
   END_RUNG
   RUNG wire#w5
      R_Coil( "Unit1.Em4.ControlNodes".cmAnodeAlignTableAxisX.commands.enableAxis )
      S_Coil( "Unit1.Em4.HmiInterface".cmAnodeAlignTableAxisX.commands.enableAxis )
   END_RUNG
   RUNG wire#w5
      R_Coil( "Unit1.Em4.ControlNodes".cmAnodeAlignTableAxisY1.commands.enableAxis )
      S_Coil( "Unit1.Em4.HmiInterface".cmAnodeAlignTableAxisY1.commands.enableAxis )
   END_RUNG
   RUNG wire#w5
      R_Coil( "Unit1.Em4.ControlNodes".cmAnodeAlignTableAxisY2.commands.enableAxis )
      S_Coil( "Unit1.Em4.HmiInterface".cmAnodeAlignTableAxisY2.commands.enableAxis )
   END_RUNG
   RUNG wire#w1
      Contact( "Unit1.EmNodes".SS1TimeExtension )
      wire#w6
      R_Coil( "Unit1.Em4.HmiInterface".cmAnodeMainPnP1AxisX.commands.enableAxis )
      S_Coil( "Unit1.Em4.ControlNodes".cmAnodeMainPnP1AxisX.commands.enableAxis )
   END_RUNG
   RUNG wire#w6
      R_Coil( "Unit1.Em4.HmiInterface".cmAnodeMainPnP2AxisX.commands.enableAxis )
      S_Coil( "Unit1.Em4.ControlNodes".cmAnodeMainPnP2AxisX.commands.enableAxis )
   END_RUNG
   RUNG wire#w6
      R_Coil( "Unit1.Em4.HmiInterface".cmAnodeMainPnP1AxisY.commands.enableAxis )
      S_Coil( "Unit1.Em4.ControlNodes".cmAnodeMainPnP1AxisY.commands.enableAxis )
   END_RUNG
   RUNG wire#w6
      R_Coil( "Unit1.Em4.HmiInterface".cmAnodeMainPnP1AxisZ.commands.enableAxis )
      S_Coil( "Unit1.Em4.ControlNodes".cmAnodeMainPnP1AxisZ.commands.enableAxis )
   END_RUNG
   RUNG wire#w6
      R_Coil( "Unit1.Em4.HmiInterface".cmAnodeMainPnP2AxisZ.commands.enableAxis )
      S_Coil( "Unit1.Em4.ControlNodes".cmAnodeMainPnP2AxisZ.commands.enableAxis )
   END_RUNG
   RUNG wire#w6
      R_Coil( "Unit1.Em4.HmiInterface".cmAnodeAlignTableAxisX.commands.enableAxis )
      S_Coil( "Unit1.Em4.ControlNodes".cmAnodeAlignTableAxisX.commands.enableAxis )
   END_RUNG
   RUNG wire#w6
      R_Coil( "Unit1.Em4.HmiInterface".cmAnodeAlignTableAxisY1.commands.enableAxis )
      S_Coil( "Unit1.Em4.ControlNodes".cmAnodeAlignTableAxisY1.commands.enableAxis )
   END_RUNG
   RUNG wire#w6
      R_Coil( "Unit1.Em4.HmiInterface".cmAnodeAlignTableAxisY2.commands.enableAxis )
      S_Coil( "Unit1.Em4.ControlNodes".cmAnodeAlignTableAxisY2.commands.enableAxis )
   END_RUNG
   RUNG wire#powerrail
      Contact( "Unit1.EmNodes".AllSFDoorOpen )
      I_Contact( "Unit1.EmNodes".SS1TimeExtension )
      I_Contact( "Unit1.EmNodes".scsMode.auto )
      wire#w7
      Contact( "Unit1.EmNodes".MobilePanelPermissions )
      I_Contact( "Unit1.EmNodes".pHmiMode.enable )
      wire#w8
      Contact( #statSlmStatus.running )
      P_Trig( #statPulse.axisEnable[5] )
      wire#w9
      R_Coil( "Unit1.Em4.ControlNodes".cmAnodeMainPnP1AxisX.commands.enableAxis )
      R_Coil( "Unit1.Em4.HmiInterface".cmAnodeMainPnP1AxisX.commands.enableAxis )
   END_RUNG
   RUNG wire#w7
      I_Contact( "Unit1.EmNodes".MobilePanelPermissions )
      I_Contact( "Unit1.EmNodes".mainOpMode.enable )
   END_RUNG wire#w8
   RUNG wire#w9
      R_Coil( "Unit1.Em4.ControlNodes".cmAnodeMainPnP2AxisX.commands.enableAxis )
      R_Coil( "Unit1.Em4.HmiInterface".cmAnodeMainPnP2AxisX.commands.enableAxis )
   END_RUNG
   RUNG wire#w9
      R_Coil( "Unit1.Em4.ControlNodes".cmAnodeMainPnP1AxisY.commands.enableAxis )
      R_Coil( "Unit1.Em4.HmiInterface".cmAnodeMainPnP1AxisY.commands.enableAxis )
   END_RUNG
   RUNG wire#w9
      R_Coil( "Unit1.Em4.ControlNodes".cmAnodeMainPnP1AxisZ.commands.enableAxis )
      R_Coil( "Unit1.Em4.HmiInterface".cmAnodeMainPnP1AxisZ.commands.enableAxis )
   END_RUNG
   RUNG wire#w9
      R_Coil( "Unit1.Em4.ControlNodes".cmAnodeMainPnP2AxisZ.commands.enableAxis )
      R_Coil( "Unit1.Em4.HmiInterface".cmAnodeMainPnP2AxisZ.commands.enableAxis )
   END_RUNG
   RUNG wire#w9
      R_Coil( "Unit1.Em4.ControlNodes".cmAnodeAlignTableAxisX.commands.enableAxis )
      R_Coil( "Unit1.Em4.HmiInterface".cmAnodeAlignTableAxisX.commands.enableAxis )
   END_RUNG
   RUNG wire#w9
      R_Coil( "Unit1.Em4.ControlNodes".cmAnodeAlignTableAxisY1.commands.enableAxis )
      R_Coil( "Unit1.Em4.HmiInterface".cmAnodeAlignTableAxisY1.commands.enableAxis )
   END_RUNG
   RUNG wire#w9
      R_Coil( "Unit1.Em4.ControlNodes".cmAnodeAlignTableAxisY2.commands.enableAxis )
      R_Coil( "Unit1.Em4.HmiInterface".cmAnodeAlignTableAxisY2.commands.enableAxis )
   END_RUNG
   // the same network as SCL:
   #_w1 := "Unit1.EmNodes".AllSFDoorOpen AND ("Unit1.EmNodes".pHmiMode.enable OR (NOT "Unit1.EmNodes".MobilePanelPermissions AND "Unit1.EmNodes".mainOpMode.enable)) AND #statSlmStatus.running;
   #_w2 := #_w1 AND NOT #statPulse.axisEnable[4];   // rising edge
   #statPulse.axisEnable[4] := #_w1;
   IF #_w2 AND #statUnitStatus.mode.production THEN
       "Unit1.Em4.HmiInterface".cmAnodeMainPnP1AxisX.commands.enableAxis := FALSE;
       "Unit1.Em4.ControlNodes".cmAnodeMainPnP1AxisX.commands.enableAxis := TRUE;
       "Unit1.Em4.HmiInterface".cmAnodeMainPnP2AxisX.commands.enableAxis := FALSE;
       "Unit1.Em4.ControlNodes".cmAnodeMainPnP2AxisX.commands.enableAxis := TRUE;
       "Unit1.Em4.HmiInterface".cmAnodeMainPnP1AxisY.commands.enableAxis := FALSE;
       "Unit1.Em4.ControlNodes".cmAnodeMainPnP1AxisY.commands.enableAxis := TRUE;
       "Unit1.Em4.HmiInterface".cmAnodeMainPnP1AxisZ.commands.enableAxis := FALSE;
       "Unit1.Em4.ControlNodes".cmAnodeMainPnP1AxisZ.commands.enableAxis := TRUE;
       "Unit1.Em4.HmiInterface".cmAnodeMainPnP2AxisZ.commands.enableAxis := FALSE;
       "Unit1.Em4.ControlNodes".cmAnodeMainPnP2AxisZ.commands.enableAxis := TRUE;
       "Unit1.Em4.HmiInterface".cmAnodeAlignTableAxisX.commands.enableAxis := FALSE;
       "Unit1.Em4.ControlNodes".cmAnodeAlignTableAxisX.commands.enableAxis := TRUE;
       "Unit1.Em4.HmiInterface".cmAnodeAlignTableAxisY1.commands.enableAxis := FALSE;
       "Unit1.Em4.ControlNodes".cmAnodeAlignTableAxisY1.commands.enableAxis := TRUE;
       "Unit1.Em4.HmiInterface".cmAnodeAlignTableAxisY2.commands.enableAxis := FALSE;
       "Unit1.Em4.ControlNodes".cmAnodeAlignTableAxisY2.commands.enableAxis := TRUE;
   END_IF;
   IF #_w2 AND (#statUnitStatus.mode.manual OR #statUnitStatus.mode.maintenance) THEN
       "Unit1.Em4.ControlNodes".cmAnodeMainPnP1AxisX.commands.enableAxis := FALSE;
       "Unit1.Em4.HmiInterface".cmAnodeMainPnP1AxisX.commands.enableAxis := TRUE;
       "Unit1.Em4.ControlNodes".cmAnodeMainPnP2AxisX.commands.enableAxis := FALSE;
       "Unit1.Em4.HmiInterface".cmAnodeMainPnP2AxisX.commands.enableAxis := TRUE;
       "Unit1.Em4.ControlNodes".cmAnodeMainPnP1AxisY.commands.enableAxis := FALSE;
       "Unit1.Em4.HmiInterface".cmAnodeMainPnP1AxisY.commands.enableAxis := TRUE;
       "Unit1.Em4.ControlNodes".cmAnodeMainPnP1AxisZ.commands.enableAxis := FALSE;
       "Unit1.Em4.HmiInterface".cmAnodeMainPnP1AxisZ.commands.enableAxis := TRUE;
       "Unit1.Em4.ControlNodes".cmAnodeMainPnP2AxisZ.commands.enableAxis := FALSE;
       "Unit1.Em4.HmiInterface".cmAnodeMainPnP2AxisZ.commands.enableAxis := TRUE;
       "Unit1.Em4.ControlNodes".cmAnodeAlignTableAxisX.commands.enableAxis := FALSE;
       "Unit1.Em4.HmiInterface".cmAnodeAlignTableAxisX.commands.enableAxis := TRUE;
       "Unit1.Em4.ControlNodes".cmAnodeAlignTableAxisY1.commands.enableAxis := FALSE;
       "Unit1.Em4.HmiInterface".cmAnodeAlignTableAxisY1.commands.enableAxis := TRUE;
       "Unit1.Em4.ControlNodes".cmAnodeAlignTableAxisY2.commands.enableAxis := FALSE;
       "Unit1.Em4.HmiInterface".cmAnodeAlignTableAxisY2.commands.enableAxis := TRUE;
   END_IF;
   IF "Unit1.EmNodes".AllSFDoorOpen AND "Unit1.EmNodes".SS1TimeExtension THEN
       "Unit1.Em4.HmiInterface".cmAnodeMainPnP1AxisX.commands.enableAxis := FALSE;
       "Unit1.Em4.ControlNodes".cmAnodeMainPnP1AxisX.commands.enableAxis := TRUE;
       "Unit1.Em4.HmiInterface".cmAnodeMainPnP2AxisX.commands.enableAxis := FALSE;
       "Unit1.Em4.ControlNodes".cmAnodeMainPnP2AxisX.commands.enableAxis := TRUE;
       "Unit1.Em4.HmiInterface".cmAnodeMainPnP1AxisY.commands.enableAxis := FALSE;
       "Unit1.Em4.ControlNodes".cmAnodeMainPnP1AxisY.commands.enableAxis := TRUE;
       "Unit1.Em4.HmiInterface".cmAnodeMainPnP1AxisZ.commands.enableAxis := FALSE;
       "Unit1.Em4.ControlNodes".cmAnodeMainPnP1AxisZ.commands.enableAxis := TRUE;
       "Unit1.Em4.HmiInterface".cmAnodeMainPnP2AxisZ.commands.enableAxis := FALSE;
       "Unit1.Em4.ControlNodes".cmAnodeMainPnP2AxisZ.commands.enableAxis := TRUE;
       "Unit1.Em4.HmiInterface".cmAnodeAlignTableAxisX.commands.enableAxis := FALSE;
       "Unit1.Em4.ControlNodes".cmAnodeAlignTableAxisX.commands.enableAxis := TRUE;
       "Unit1.Em4.HmiInterface".cmAnodeAlignTableAxisY1.commands.enableAxis := FALSE;
       "Unit1.Em4.ControlNodes".cmAnodeAlignTableAxisY1.commands.enableAxis := TRUE;
       "Unit1.Em4.HmiInterface".cmAnodeAlignTableAxisY2.commands.enableAxis := FALSE;
       "Unit1.Em4.ControlNodes".cmAnodeAlignTableAxisY2.commands.enableAxis := TRUE;
   END_IF;
   #_w3 := "Unit1.EmNodes".AllSFDoorOpen AND NOT "Unit1.EmNodes".SS1TimeExtension AND NOT "Unit1.EmNodes".scsMode.auto AND (("Unit1.EmNodes".MobilePanelPermissions AND NOT "Unit1.EmNodes".pHmiMode.enable) OR (NOT "Unit1.EmNodes".MobilePanelPermissions AND NOT "Unit1.EmNodes".mainOpMode.enable)) AND #statSlmStatus.running;
   #_w4 := #_w3 AND NOT #statPulse.axisEnable[5];   // rising edge
   #statPulse.axisEnable[5] := #_w3;
   IF #_w4 THEN
       "Unit1.Em4.ControlNodes".cmAnodeMainPnP1AxisX.commands.enableAxis := FALSE;
       "Unit1.Em4.HmiInterface".cmAnodeMainPnP1AxisX.commands.enableAxis := FALSE;
       "Unit1.Em4.ControlNodes".cmAnodeMainPnP2AxisX.commands.enableAxis := FALSE;
       "Unit1.Em4.HmiInterface".cmAnodeMainPnP2AxisX.commands.enableAxis := FALSE;
       "Unit1.Em4.ControlNodes".cmAnodeMainPnP1AxisY.commands.enableAxis := FALSE;
       "Unit1.Em4.HmiInterface".cmAnodeMainPnP1AxisY.commands.enableAxis := FALSE;
       "Unit1.Em4.ControlNodes".cmAnodeMainPnP1AxisZ.commands.enableAxis := FALSE;
       "Unit1.Em4.HmiInterface".cmAnodeMainPnP1AxisZ.commands.enableAxis := FALSE;
       "Unit1.Em4.ControlNodes".cmAnodeMainPnP2AxisZ.commands.enableAxis := FALSE;
       "Unit1.Em4.HmiInterface".cmAnodeMainPnP2AxisZ.commands.enableAxis := FALSE;
       "Unit1.Em4.ControlNodes".cmAnodeAlignTableAxisX.commands.enableAxis := FALSE;
       "Unit1.Em4.HmiInterface".cmAnodeAlignTableAxisX.commands.enableAxis := FALSE;
       "Unit1.Em4.ControlNodes".cmAnodeAlignTableAxisY1.commands.enableAxis := FALSE;
       "Unit1.Em4.HmiInterface".cmAnodeAlignTableAxisY1.commands.enableAxis := FALSE;
       "Unit1.Em4.ControlNodes".cmAnodeAlignTableAxisY2.commands.enableAxis := FALSE;
       "Unit1.Em4.HmiInterface".cmAnodeAlignTableAxisY2.commands.enableAxis := FALSE;
   END_IF;
END_REGION

REGION Network 80: Disable All CMs
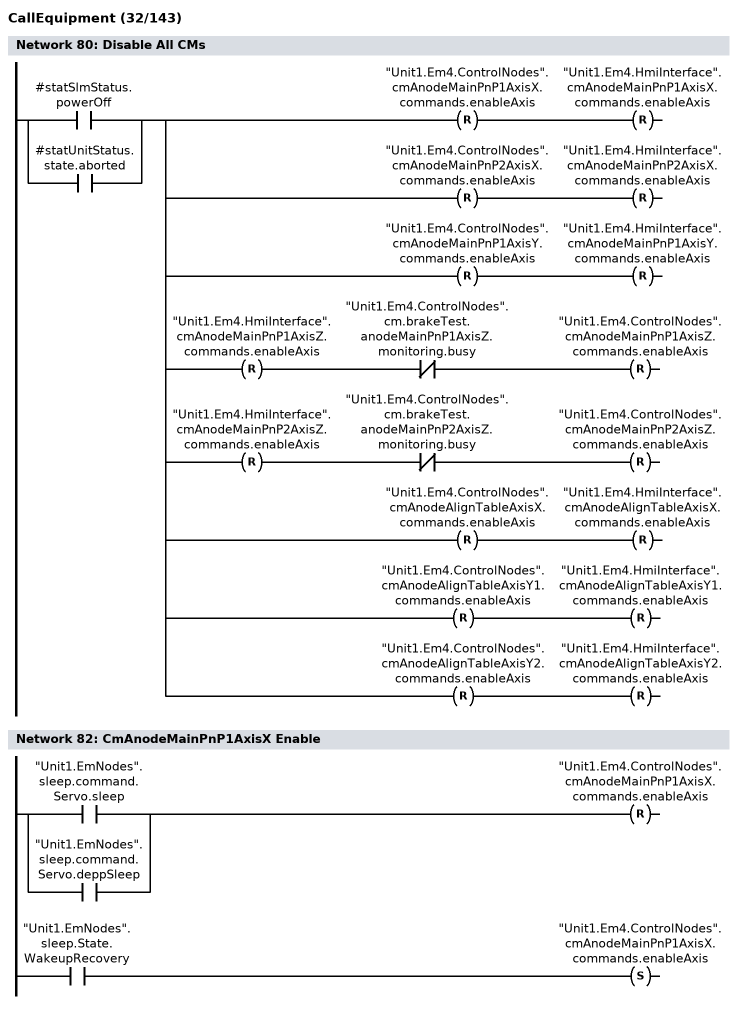
   RUNG wire#powerrail
      Contact( #statSlmStatus.powerOff )
      wire#w1
      R_Coil( "Unit1.Em4.ControlNodes".cmAnodeMainPnP1AxisX.commands.enableAxis )
      R_Coil( "Unit1.Em4.HmiInterface".cmAnodeMainPnP1AxisX.commands.enableAxis )
   END_RUNG
   RUNG wire#powerrail
      Contact( #statUnitStatus.state.aborted )
   END_RUNG wire#w1
   RUNG wire#w1
      R_Coil( "Unit1.Em4.ControlNodes".cmAnodeMainPnP2AxisX.commands.enableAxis )
      R_Coil( "Unit1.Em4.HmiInterface".cmAnodeMainPnP2AxisX.commands.enableAxis )
   END_RUNG
   RUNG wire#w1
      R_Coil( "Unit1.Em4.ControlNodes".cmAnodeMainPnP1AxisY.commands.enableAxis )
      R_Coil( "Unit1.Em4.HmiInterface".cmAnodeMainPnP1AxisY.commands.enableAxis )
   END_RUNG
   RUNG wire#w1
      R_Coil( "Unit1.Em4.HmiInterface".cmAnodeMainPnP1AxisZ.commands.enableAxis )
      I_Contact( "Unit1.Em4.ControlNodes".cm.brakeTest.anodeMainPnP1AxisZ.monitoring.busy )
      R_Coil( "Unit1.Em4.ControlNodes".cmAnodeMainPnP1AxisZ.commands.enableAxis )
   END_RUNG
   RUNG wire#w1
      R_Coil( "Unit1.Em4.HmiInterface".cmAnodeMainPnP2AxisZ.commands.enableAxis )
      I_Contact( "Unit1.Em4.ControlNodes".cm.brakeTest.anodeMainPnP2AxisZ.monitoring.busy )
      R_Coil( "Unit1.Em4.ControlNodes".cmAnodeMainPnP2AxisZ.commands.enableAxis )
   END_RUNG
   RUNG wire#w1
      R_Coil( "Unit1.Em4.ControlNodes".cmAnodeAlignTableAxisX.commands.enableAxis )
      R_Coil( "Unit1.Em4.HmiInterface".cmAnodeAlignTableAxisX.commands.enableAxis )
   END_RUNG
   RUNG wire#w1
      R_Coil( "Unit1.Em4.ControlNodes".cmAnodeAlignTableAxisY1.commands.enableAxis )
      R_Coil( "Unit1.Em4.HmiInterface".cmAnodeAlignTableAxisY1.commands.enableAxis )
   END_RUNG
   RUNG wire#w1
      R_Coil( "Unit1.Em4.ControlNodes".cmAnodeAlignTableAxisY2.commands.enableAxis )
      R_Coil( "Unit1.Em4.HmiInterface".cmAnodeAlignTableAxisY2.commands.enableAxis )
   END_RUNG
   // the same network as SCL:
   #_w1 := #statSlmStatus.powerOff OR #statUnitStatus.state.aborted;
   IF #_w1 THEN
       "Unit1.Em4.ControlNodes".cmAnodeMainPnP1AxisX.commands.enableAxis := FALSE;
       "Unit1.Em4.HmiInterface".cmAnodeMainPnP1AxisX.commands.enableAxis := FALSE;
       "Unit1.Em4.ControlNodes".cmAnodeMainPnP2AxisX.commands.enableAxis := FALSE;
       "Unit1.Em4.HmiInterface".cmAnodeMainPnP2AxisX.commands.enableAxis := FALSE;
       "Unit1.Em4.ControlNodes".cmAnodeMainPnP1AxisY.commands.enableAxis := FALSE;
       "Unit1.Em4.HmiInterface".cmAnodeMainPnP1AxisY.commands.enableAxis := FALSE;
       "Unit1.Em4.HmiInterface".cmAnodeMainPnP1AxisZ.commands.enableAxis := FALSE;
   END_IF;
   IF #_w1 AND NOT "Unit1.Em4.ControlNodes".cm.brakeTest.anodeMainPnP1AxisZ.monitoring.busy THEN
       "Unit1.Em4.ControlNodes".cmAnodeMainPnP1AxisZ.commands.enableAxis := FALSE;
   END_IF;
   IF #_w1 THEN "Unit1.Em4.HmiInterface".cmAnodeMainPnP2AxisZ.commands.enableAxis := FALSE; END_IF;
   IF #_w1 AND NOT "Unit1.Em4.ControlNodes".cm.brakeTest.anodeMainPnP2AxisZ.monitoring.busy THEN
       "Unit1.Em4.ControlNodes".cmAnodeMainPnP2AxisZ.commands.enableAxis := FALSE;
   END_IF;
   IF #_w1 THEN
       "Unit1.Em4.ControlNodes".cmAnodeAlignTableAxisX.commands.enableAxis := FALSE;
       "Unit1.Em4.HmiInterface".cmAnodeAlignTableAxisX.commands.enableAxis := FALSE;
       "Unit1.Em4.ControlNodes".cmAnodeAlignTableAxisY1.commands.enableAxis := FALSE;
       "Unit1.Em4.HmiInterface".cmAnodeAlignTableAxisY1.commands.enableAxis := FALSE;
       "Unit1.Em4.ControlNodes".cmAnodeAlignTableAxisY2.commands.enableAxis := FALSE;
       "Unit1.Em4.HmiInterface".cmAnodeAlignTableAxisY2.commands.enableAxis := FALSE;
   END_IF;
END_REGION

REGION Network 82: CmAnodeMainPnP1AxisX Enable
   RUNG wire#powerrail
      Contact( "Unit1.EmNodes".sleep.command.Servo.sleep )
      wire#w1
      R_Coil( "Unit1.Em4.ControlNodes".cmAnodeMainPnP1AxisX.commands.enableAxis )
   END_RUNG
   RUNG wire#powerrail
      Contact( "Unit1.EmNodes".sleep.command.Servo.deppSleep )
   END_RUNG wire#w1
   RUNG wire#powerrail
      Contact( "Unit1.EmNodes".sleep.State.WakeupRecovery )
      S_Coil( "Unit1.Em4.ControlNodes".cmAnodeMainPnP1AxisX.commands.enableAxis )
   END_RUNG
   // the same network as SCL:
   IF "Unit1.EmNodes".sleep.command.Servo.sleep OR "Unit1.EmNodes".sleep.command.Servo.deppSleep THEN
       "Unit1.Em4.ControlNodes".cmAnodeMainPnP1AxisX.commands.enableAxis := FALSE;
   END_IF;
   IF "Unit1.EmNodes".sleep.State.WakeupRecovery THEN
       "Unit1.Em4.ControlNodes".cmAnodeMainPnP1AxisX.commands.enableAxis := TRUE;
   END_IF;
END_REGION

REGION Network 83: Anode Main P&P 1 X-Axis Homing Interlock
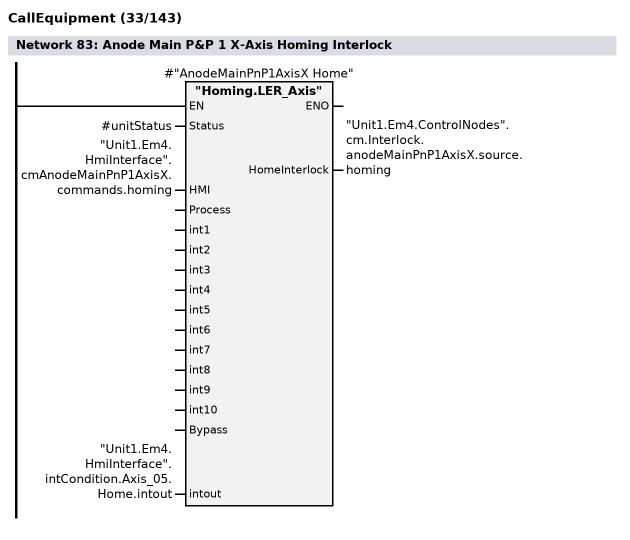
   RUNG wire#powerrail
      #"AnodeMainPnP1AxisX Home"(Status := #unitStatus, HMI := "Unit1.Em4.HmiInterface".cmAnodeMainPnP1AxisX.commands.homing, Process :=, int1 :=, int2 :=, int3 :=, int4 :=, int5 :=, int6 :=, int7 :=, int8 :=, int9 :=, int10 :=, Bypass :=, intout := "Unit1.Em4.HmiInterface".intCondition.Axis_05.Home.intout, HomeInterlock => "Unit1.Em4.ControlNodes".cm.Interlock.anodeMainPnP1AxisX.source.homing)
   END_RUNG
   // the same network as SCL:
   #"AnodeMainPnP1AxisX Home"(Status := #unitStatus,   // "Homing.LER_Axis"
                           HMI := "Unit1.Em4.HmiInterface".cmAnodeMainPnP1AxisX.commands.homing,
                           intout := "Unit1.Em4.HmiInterface".intCondition.Axis_05.Home.intout,
                           HomeInterlock => "Unit1.Em4.ControlNodes".cm.Interlock.anodeMainPnP1AxisX.source.homing);
END_REGION

REGION Network 84: CmAnodeMainPnP1AxisX Position Absolute Jog
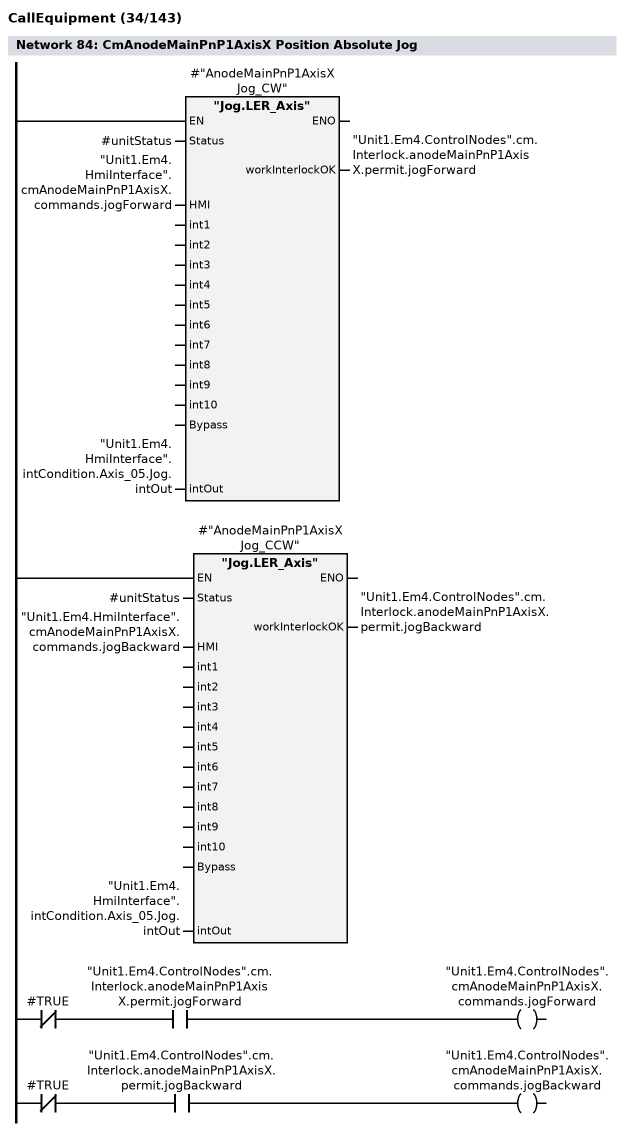
   RUNG wire#powerrail
      #"AnodeMainPnP1AxisX Jog_CW"(Status := #unitStatus, HMI := "Unit1.Em4.HmiInterface".cmAnodeMainPnP1AxisX.commands.jogForward, int1 :=, int2 :=, int3 :=, int4 :=, int5 :=, int6 :=, int7 :=, int8 :=, int9 :=, int10 :=, Bypass :=, intOut := "Unit1.Em4.HmiInterface".intCondition.Axis_05.Jog.intOut, workInterlockOK => "Unit1.Em4.ControlNodes".cm.Interlock.anodeMainPnP1AxisX.permit.jogForward)
   END_RUNG
   RUNG wire#powerrail
      #"AnodeMainPnP1AxisX Jog_CCW"(Status := #unitStatus, HMI := "Unit1.Em4.HmiInterface".cmAnodeMainPnP1AxisX.commands.jogBackward, int1 :=, int2 :=, int3 :=, int4 :=, int5 :=, int6 :=, int7 :=, int8 :=, int9 :=, int10 :=, Bypass :=, intOut := "Unit1.Em4.HmiInterface".intCondition.Axis_05.Jog.intOut, workInterlockOK => "Unit1.Em4.ControlNodes".cm.Interlock.anodeMainPnP1AxisX.permit.jogBackward)
   END_RUNG
   RUNG wire#powerrail
      I_Contact( #TRUE )
      Contact( "Unit1.Em4.ControlNodes".cm.Interlock.anodeMainPnP1AxisX.permit.jogForward )
      Coil( "Unit1.Em4.ControlNodes".cmAnodeMainPnP1AxisX.commands.jogForward )
   END_RUNG
   RUNG wire#powerrail
      I_Contact( #TRUE )
      Contact( "Unit1.Em4.ControlNodes".cm.Interlock.anodeMainPnP1AxisX.permit.jogBackward )
      Coil( "Unit1.Em4.ControlNodes".cmAnodeMainPnP1AxisX.commands.jogBackward )
   END_RUNG
   // the same network as SCL:
   #"AnodeMainPnP1AxisX Jog_CW"(Status := #unitStatus,   // "Jog.LER_Axis"
                           HMI := "Unit1.Em4.HmiInterface".cmAnodeMainPnP1AxisX.commands.jogForward,
                           intOut := "Unit1.Em4.HmiInterface".intCondition.Axis_05.Jog.intOut,
                           workInterlockOK => "Unit1.Em4.ControlNodes".cm.Interlock.anodeMainPnP1AxisX.permit.jogForward);
   #"AnodeMainPnP1AxisX Jog_CCW"(Status := #unitStatus,   // "Jog.LER_Axis"
                           HMI := "Unit1.Em4.HmiInterface".cmAnodeMainPnP1AxisX.commands.jogBackward,
                           intOut := "Unit1.Em4.HmiInterface".intCondition.Axis_05.Jog.intOut,
                           workInterlockOK => "Unit1.Em4.ControlNodes".cm.Interlock.anodeMainPnP1AxisX.permit.jogBackward);
   "Unit1.Em4.ControlNodes".cmAnodeMainPnP1AxisX.commands.jogForward := NOT #TRUE AND "Unit1.Em4.ControlNodes".cm.Interlock.anodeMainPnP1AxisX.permit.jogForward;
   "Unit1.Em4.ControlNodes".cmAnodeMainPnP1AxisX.commands.jogBackward := NOT #TRUE AND "Unit1.Em4.ControlNodes".cm.Interlock.anodeMainPnP1AxisX.permit.jogBackward;
END_REGION

REGION Network 85: CmAnodeMainPnP1AxisX Position Absolute Position0
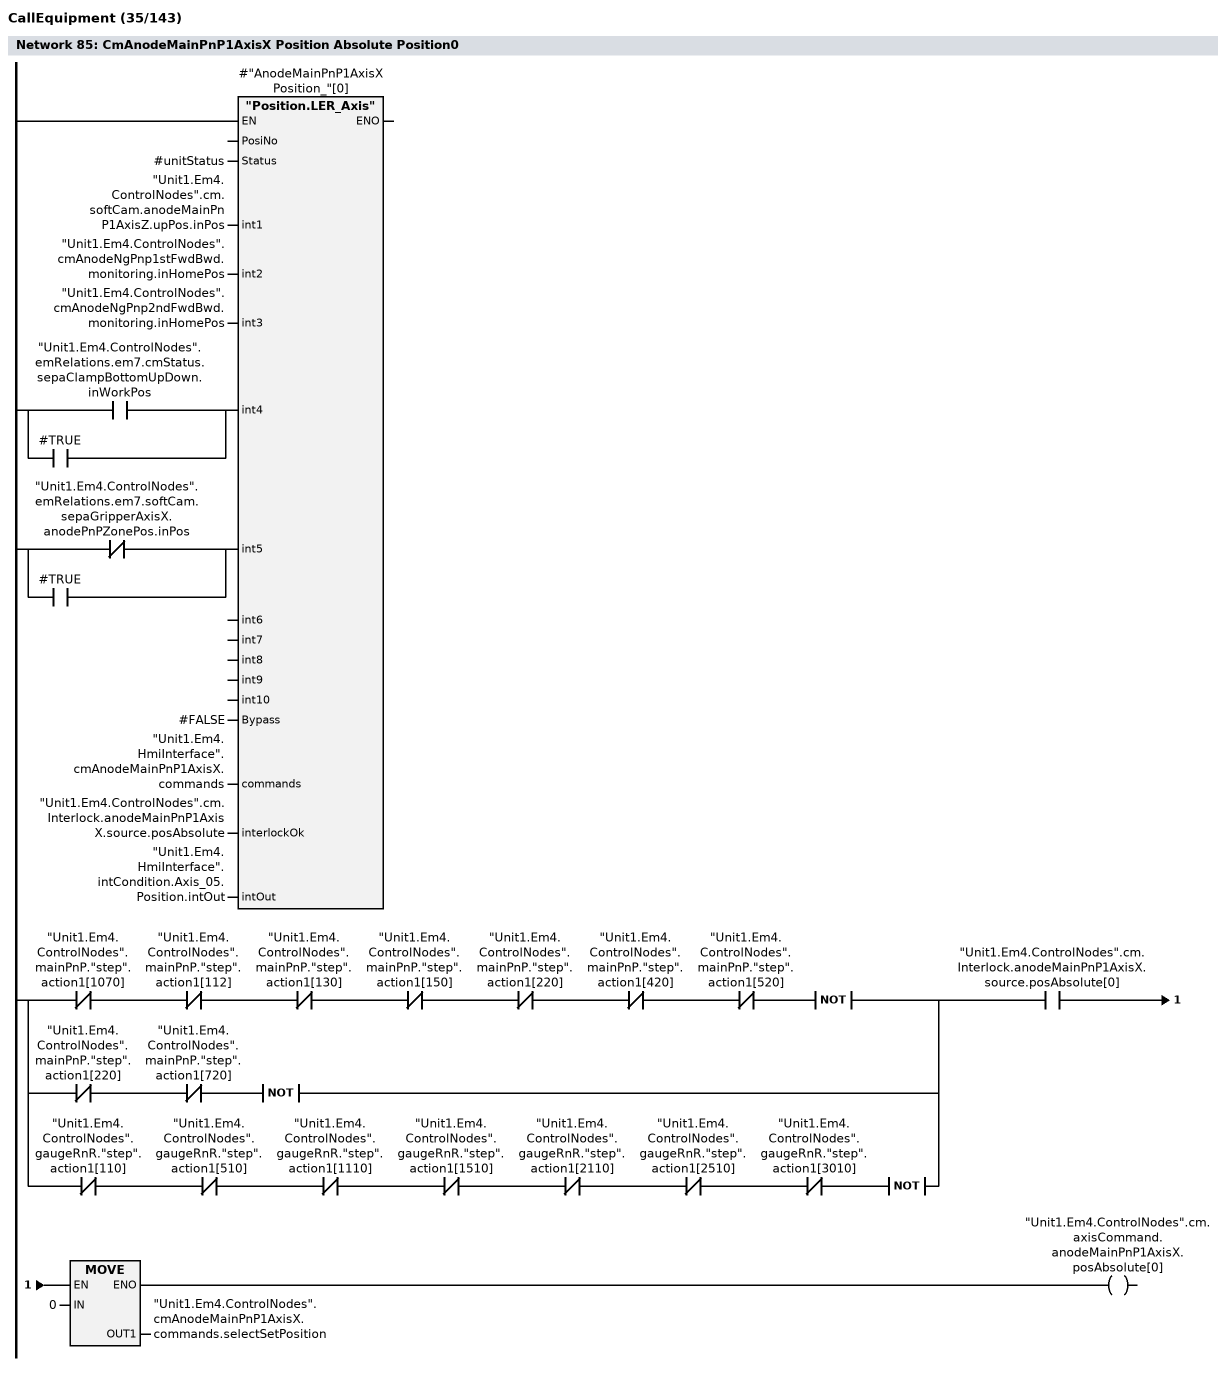
   RUNG wire#powerrail
      #"AnodeMainPnP1AxisX Position_"[0](int4 := wire#w1, int5 := wire#w2, PosiNo :=, Status := #unitStatus, int1 := "Unit1.Em4.ControlNodes".cm.softCam.anodeMainPnP1AxisZ.upPos.inPos, int2 := "Unit1.Em4.ControlNodes".cmAnodeNgPnp1stFwdBwd.monitoring.inHomePos, int3 := "Unit1.Em4.ControlNodes".cmAnodeNgPnp2ndFwdBwd.monitoring.inHomePos, int6 :=, int7 :=, int8 :=, int9 :=, int10 :=, Bypass := #FALSE, commands := "Unit1.Em4.HmiInterface".cmAnodeMainPnP1AxisX.commands, interlockOk := "Unit1.Em4.ControlNodes".cm.Interlock.anodeMainPnP1AxisX.source.posAbsolute, intOut := "Unit1.Em4.HmiInterface".intCondition.Axis_05.Position.intOut)
   END_RUNG
   RUNG wire#powerrail
      Contact( "Unit1.Em4.ControlNodes".emRelations.em7.cmStatus.sepaClampBottomUpDown.inWorkPos )
   END_RUNG wire#w1
   RUNG wire#powerrail
      Contact( #TRUE )
   END_RUNG wire#w1
   RUNG wire#powerrail
      I_Contact( "Unit1.Em4.ControlNodes".emRelations.em7.softCam.sepaGripperAxisX.anodePnPZonePos.inPos )
   END_RUNG wire#w2
   RUNG wire#powerrail
      Contact( #TRUE )
   END_RUNG wire#w2
   RUNG wire#powerrail
      I_Contact( "Unit1.Em4.ControlNodes".mainPnP."step".action1[1070] )
      I_Contact( "Unit1.Em4.ControlNodes".mainPnP."step".action1[112] )
      I_Contact( "Unit1.Em4.ControlNodes".mainPnP."step".action1[130] )
      I_Contact( "Unit1.Em4.ControlNodes".mainPnP."step".action1[150] )
      I_Contact( "Unit1.Em4.ControlNodes".mainPnP."step".action1[220] )
      I_Contact( "Unit1.Em4.ControlNodes".mainPnP."step".action1[420] )
      I_Contact( "Unit1.Em4.ControlNodes".mainPnP."step".action1[520] )
      Not()
      wire#w3
      Contact( "Unit1.Em4.ControlNodes".cm.Interlock.anodeMainPnP1AxisX.source.posAbsolute[0] )
      Move(in := 0, out1 => "Unit1.Em4.ControlNodes".cmAnodeMainPnP1AxisX.commands.selectSetPosition)
      Coil( "Unit1.Em4.ControlNodes".cm.axisCommand.anodeMainPnP1AxisX.posAbsolute[0] )
   END_RUNG
   RUNG wire#powerrail
      I_Contact( "Unit1.Em4.ControlNodes".mainPnP."step".action1[220] )
      I_Contact( "Unit1.Em4.ControlNodes".mainPnP."step".action1[720] )
      Not()
   END_RUNG wire#w3
   RUNG wire#powerrail
      I_Contact( "Unit1.Em4.ControlNodes".gaugeRnR."step".action1[110] )
      I_Contact( "Unit1.Em4.ControlNodes".gaugeRnR."step".action1[510] )
      I_Contact( "Unit1.Em4.ControlNodes".gaugeRnR."step".action1[1110] )
      I_Contact( "Unit1.Em4.ControlNodes".gaugeRnR."step".action1[1510] )
      I_Contact( "Unit1.Em4.ControlNodes".gaugeRnR."step".action1[2110] )
      I_Contact( "Unit1.Em4.ControlNodes".gaugeRnR."step".action1[2510] )
      I_Contact( "Unit1.Em4.ControlNodes".gaugeRnR."step".action1[3010] )
      Not()
   END_RUNG wire#w3
   // the same network as SCL:
   #"AnodeMainPnP1AxisX Position_"[0](Status := #unitStatus,   // "Position.LER_Axis"
                           int1 := "Unit1.Em4.ControlNodes".cm.softCam.anodeMainPnP1AxisZ.upPos.inPos,
                           int2 := "Unit1.Em4.ControlNodes".cmAnodeNgPnp1stFwdBwd.monitoring.inHomePos,
                           int3 := "Unit1.Em4.ControlNodes".cmAnodeNgPnp2ndFwdBwd.monitoring.inHomePos,
                           int4 := "Unit1.Em4.ControlNodes".emRelations.em7.cmStatus.sepaClampBottomUpDown.inWorkPos OR #TRUE,
                           int5 := NOT "Unit1.Em4.ControlNodes".emRelations.em7.softCam.sepaGripperAxisX.anodePnPZonePos.inPos OR #TRUE,
                           Bypass := #FALSE,
                           commands := "Unit1.Em4.HmiInterface".cmAnodeMainPnP1AxisX.commands,
                           interlockOk := "Unit1.Em4.ControlNodes".cm.Interlock.anodeMainPnP1AxisX.source.posAbsolute,
                           intOut := "Unit1.Em4.HmiInterface".intCondition.Axis_05.Position.intOut);
   #_w1 := (NOT (NOT "Unit1.Em4.ControlNodes".mainPnP."step".action1[1070] AND NOT "Unit1.Em4.ControlNodes".mainPnP."step".action1[112] AND NOT "Unit1.Em4.ControlNodes".mainPnP."step".action1[130] AND NOT "Unit1.Em4.ControlNodes".mainPnP."step".action1[150] AND NOT "Unit1.Em4.ControlNodes".mainPnP."step".action1[220] AND NOT "Unit1.Em4.ControlNodes".mainPnP."step".action1[420] AND NOT "Unit1.Em4.ControlNodes".mainPnP."step".action1[520]) OR NOT (NOT "Unit1.Em4.ControlNodes".mainPnP."step".action1[220] AND NOT "Unit1.Em4.ControlNodes".mainPnP."step".action1[720]) OR NOT (NOT "Unit1.Em4.ControlNodes".gaugeRnR."step".action1[110] AND NOT "Unit1.Em4.ControlNodes".gaugeRnR."step".action1[510] AND NOT "Unit1.Em4.ControlNodes".gaugeRnR."step".action1[1110] AND NOT "Unit1.Em4.ControlNodes".gaugeRnR."step".action1[1510] AND NOT "Unit1.Em4.ControlNodes".gaugeRnR."step".action1[2110] AND NOT "Unit1.Em4.ControlNodes".gaugeRnR."step".action1[2510] AND NOT "Unit1.Em4.ControlNodes".gaugeRnR."step".action1[3010])) AND "Unit1.Em4.ControlNodes".cm.Interlock.anodeMainPnP1AxisX.source.posAbsolute[0];
   IF #_w1 THEN "Unit1.Em4.ControlNodes".cmAnodeMainPnP1AxisX.commands.selectSetPosition := 0; END_IF;
   "Unit1.Em4.ControlNodes".cm.axisCommand.anodeMainPnP1AxisX.posAbsolute[0] := #_w1;
END_REGION

REGION Network 86: CmAnodeMainPnP1AxisX Position Absolute Position1
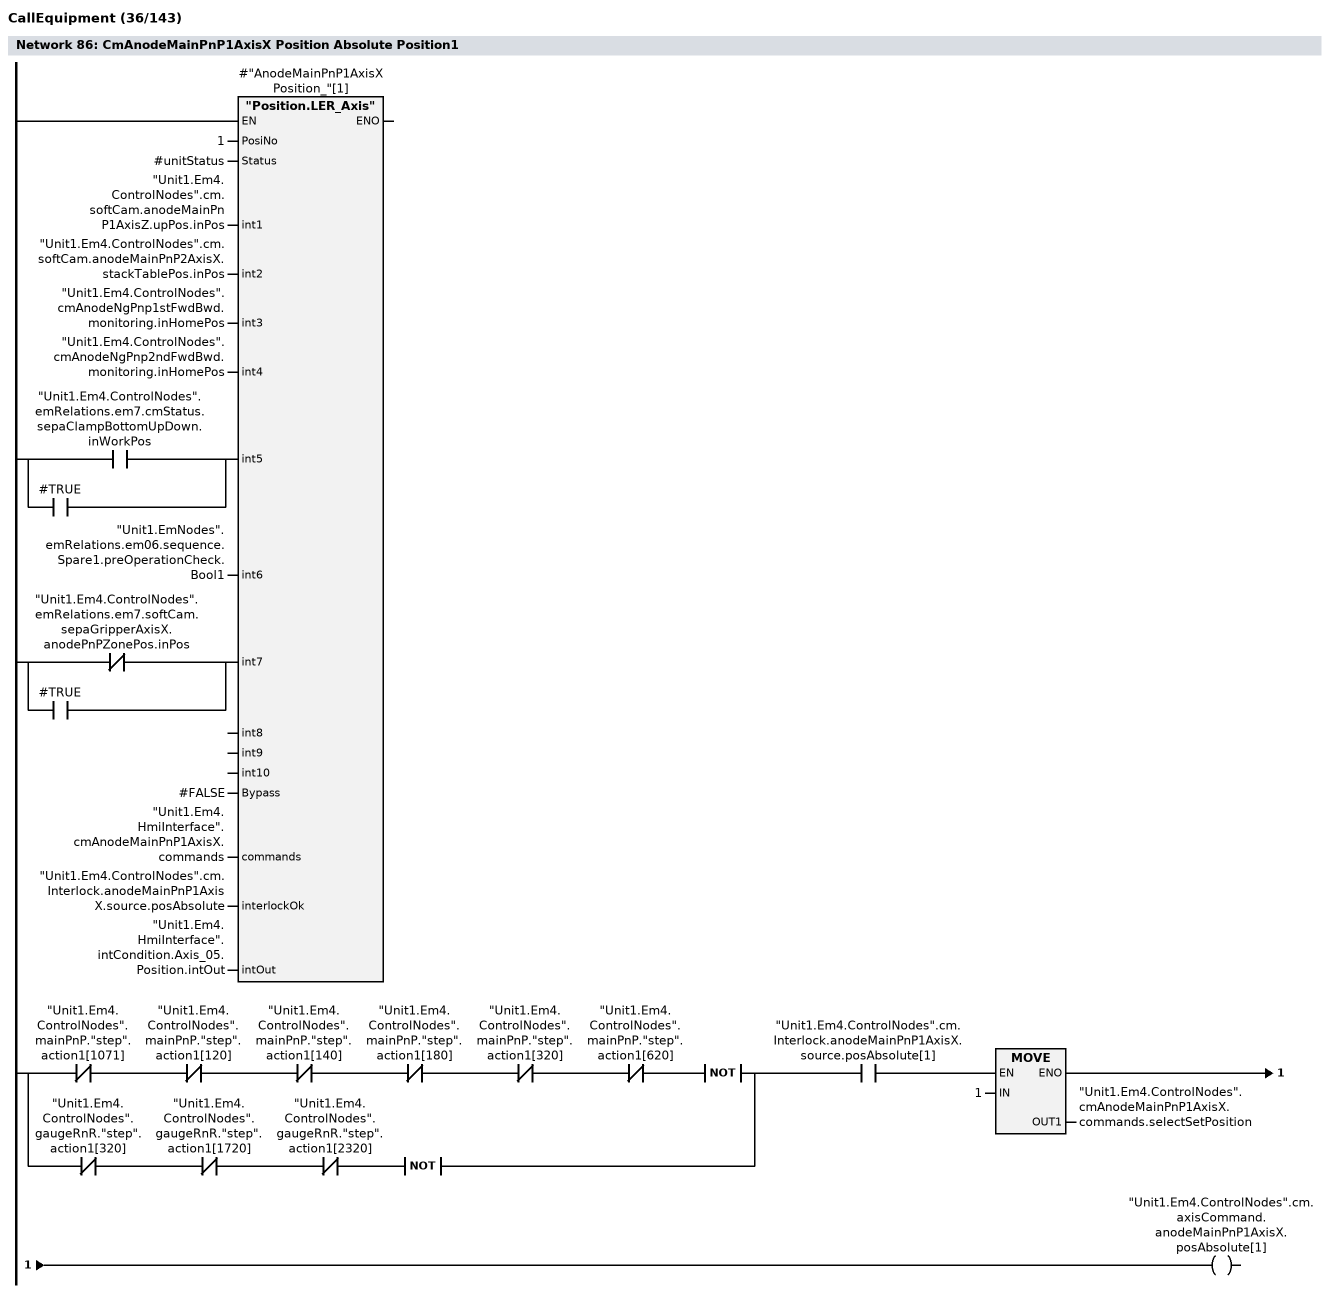
   RUNG wire#powerrail
      #"AnodeMainPnP1AxisX Position_"[1](int5 := wire#w1, int7 := wire#w2, PosiNo := 1, Status := #unitStatus, int1 := "Unit1.Em4.ControlNodes".cm.softCam.anodeMainPnP1AxisZ.upPos.inPos, int2 := "Unit1.Em4.ControlNodes".cm.softCam.anodeMainPnP2AxisX.stackTablePos.inPos, int3 := "Unit1.Em4.ControlNodes".cmAnodeNgPnp1stFwdBwd.monitoring.inHomePos, int4 := "Unit1.Em4.ControlNodes".cmAnodeNgPnp2ndFwdBwd.monitoring.inHomePos, int6 := "Unit1.EmNodes".emRelations.em06.sequence.Spare1.preOperationCheck.Bool1, int8 :=, int9 :=, int10 :=, Bypass := #FALSE, commands := "Unit1.Em4.HmiInterface".cmAnodeMainPnP1AxisX.commands, interlockOk := "Unit1.Em4.ControlNodes".cm.Interlock.anodeMainPnP1AxisX.source.posAbsolute, intOut := "Unit1.Em4.HmiInterface".intCondition.Axis_05.Position.intOut)
   END_RUNG
   RUNG wire#powerrail
      Contact( "Unit1.Em4.ControlNodes".emRelations.em7.cmStatus.sepaClampBottomUpDown.inWorkPos )
   END_RUNG wire#w1
   RUNG wire#powerrail
      Contact( #TRUE )
   END_RUNG wire#w1
   RUNG wire#powerrail
      I_Contact( "Unit1.Em4.ControlNodes".emRelations.em7.softCam.sepaGripperAxisX.anodePnPZonePos.inPos )
   END_RUNG wire#w2
   RUNG wire#powerrail
      Contact( #TRUE )
   END_RUNG wire#w2
   RUNG wire#powerrail
      I_Contact( "Unit1.Em4.ControlNodes".mainPnP."step".action1[1071] )
      I_Contact( "Unit1.Em4.ControlNodes".mainPnP."step".action1[120] )
      I_Contact( "Unit1.Em4.ControlNodes".mainPnP."step".action1[140] )
      I_Contact( "Unit1.Em4.ControlNodes".mainPnP."step".action1[180] )
      I_Contact( "Unit1.Em4.ControlNodes".mainPnP."step".action1[320] )
      I_Contact( "Unit1.Em4.ControlNodes".mainPnP."step".action1[620] )
      Not()
      wire#w3
      Contact( "Unit1.Em4.ControlNodes".cm.Interlock.anodeMainPnP1AxisX.source.posAbsolute[1] )
      Move(in := 1, out1 => "Unit1.Em4.ControlNodes".cmAnodeMainPnP1AxisX.commands.selectSetPosition)
      Coil( "Unit1.Em4.ControlNodes".cm.axisCommand.anodeMainPnP1AxisX.posAbsolute[1] )
   END_RUNG
   RUNG wire#powerrail
      I_Contact( "Unit1.Em4.ControlNodes".gaugeRnR."step".action1[320] )
      I_Contact( "Unit1.Em4.ControlNodes".gaugeRnR."step".action1[1720] )
      I_Contact( "Unit1.Em4.ControlNodes".gaugeRnR."step".action1[2320] )
      Not()
   END_RUNG wire#w3
   // the same network as SCL:
   #"AnodeMainPnP1AxisX Position_"[1](PosiNo := 1,   // "Position.LER_Axis"
                           Status := #unitStatus,
                           int1 := "Unit1.Em4.ControlNodes".cm.softCam.anodeMainPnP1AxisZ.upPos.inPos,
                           int2 := "Unit1.Em4.ControlNodes".cm.softCam.anodeMainPnP2AxisX.stackTablePos.inPos,
                           int3 := "Unit1.Em4.ControlNodes".cmAnodeNgPnp1stFwdBwd.monitoring.inHomePos,
                           int4 := "Unit1.Em4.ControlNodes".cmAnodeNgPnp2ndFwdBwd.monitoring.inHomePos,
                           int5 := "Unit1.Em4.ControlNodes".emRelations.em7.cmStatus.sepaClampBottomUpDown.inWorkPos OR #TRUE,
                           int6 := "Unit1.EmNodes".emRelations.em06.sequence.Spare1.preOperationCheck.Bool1,
                           int7 := NOT "Unit1.Em4.ControlNodes".emRelations.em7.softCam.sepaGripperAxisX.anodePnPZonePos.inPos OR #TRUE,
                           Bypass := #FALSE,
                           commands := "Unit1.Em4.HmiInterface".cmAnodeMainPnP1AxisX.commands,
                           interlockOk := "Unit1.Em4.ControlNodes".cm.Interlock.anodeMainPnP1AxisX.source.posAbsolute,
                           intOut := "Unit1.Em4.HmiInterface".intCondition.Axis_05.Position.intOut);
   #_w1 := (NOT (NOT "Unit1.Em4.ControlNodes".mainPnP."step".action1[1071] AND NOT "Unit1.Em4.ControlNodes".mainPnP."step".action1[120] AND NOT "Unit1.Em4.ControlNodes".mainPnP."step".action1[140] AND NOT "Unit1.Em4.ControlNodes".mainPnP."step".action1[180] AND NOT "Unit1.Em4.ControlNodes".mainPnP."step".action1[320] AND NOT "Unit1.Em4.ControlNodes".mainPnP."step".action1[620]) OR NOT (NOT "Unit1.Em4.ControlNodes".gaugeRnR."step".action1[320] AND NOT "Unit1.Em4.ControlNodes".gaugeRnR."step".action1[1720] AND NOT "Unit1.Em4.ControlNodes".gaugeRnR."step".action1[2320])) AND "Unit1.Em4.ControlNodes".cm.Interlock.anodeMainPnP1AxisX.source.posAbsolute[1];
   IF #_w1 THEN "Unit1.Em4.ControlNodes".cmAnodeMainPnP1AxisX.commands.selectSetPosition := 1; END_IF;
   "Unit1.Em4.ControlNodes".cm.axisCommand.anodeMainPnP1AxisX.posAbsolute[1] := #_w1;
END_REGION

REGION Network 87: CmAnodeMainPnP1AxisX Position Absolute Position2
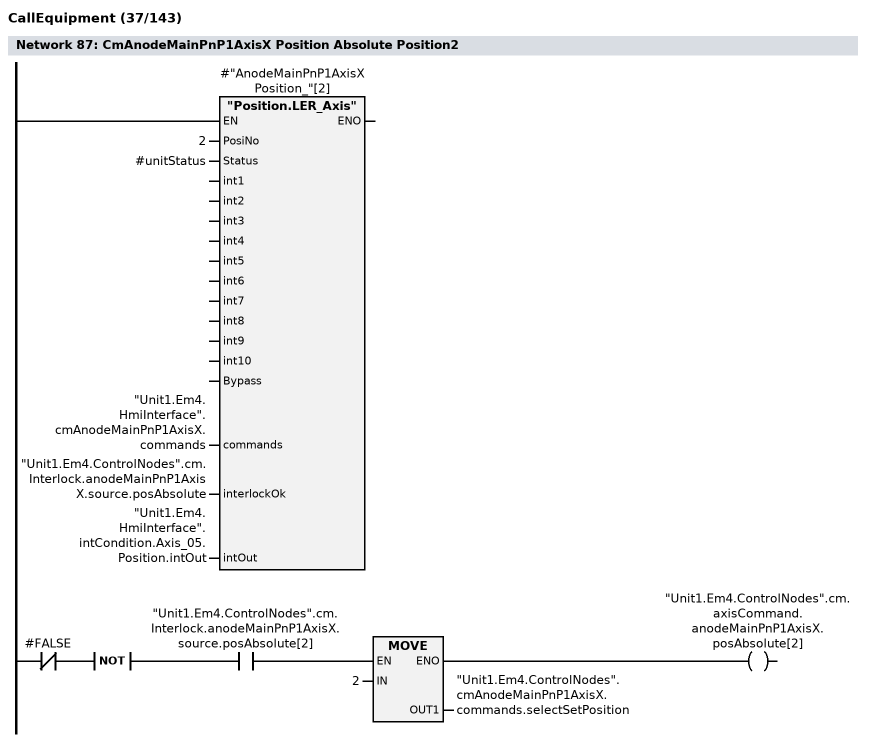
   RUNG wire#powerrail
      #"AnodeMainPnP1AxisX Position_"[2](PosiNo := 2, Status := #unitStatus, int1 :=, int2 :=, int3 :=, int4 :=, int5 :=, int6 :=, int7 :=, int8 :=, int9 :=, int10 :=, Bypass :=, commands := "Unit1.Em4.HmiInterface".cmAnodeMainPnP1AxisX.commands, interlockOk := "Unit1.Em4.ControlNodes".cm.Interlock.anodeMainPnP1AxisX.source.posAbsolute, intOut := "Unit1.Em4.HmiInterface".intCondition.Axis_05.Position.intOut)
   END_RUNG
   RUNG wire#powerrail
      I_Contact( #FALSE )
      Not()
      Contact( "Unit1.Em4.ControlNodes".cm.Interlock.anodeMainPnP1AxisX.source.posAbsolute[2] )
      Move(in := 2, out1 => "Unit1.Em4.ControlNodes".cmAnodeMainPnP1AxisX.commands.selectSetPosition)
      Coil( "Unit1.Em4.ControlNodes".cm.axisCommand.anodeMainPnP1AxisX.posAbsolute[2] )
   END_RUNG
   // the same network as SCL:
   #"AnodeMainPnP1AxisX Position_"[2](PosiNo := 2,   // "Position.LER_Axis"
                           Status := #unitStatus,
                           commands := "Unit1.Em4.HmiInterface".cmAnodeMainPnP1AxisX.commands,
                           interlockOk := "Unit1.Em4.ControlNodes".cm.Interlock.anodeMainPnP1AxisX.source.posAbsolute,
                           intOut := "Unit1.Em4.HmiInterface".intCondition.Axis_05.Position.intOut);
   #_w1 := NOT (NOT #FALSE) AND "Unit1.Em4.ControlNodes".cm.Interlock.anodeMainPnP1AxisX.source.posAbsolute[2];
   IF #_w1 THEN "Unit1.Em4.ControlNodes".cmAnodeMainPnP1AxisX.commands.selectSetPosition := 2; END_IF;
   "Unit1.Em4.ControlNodes".cm.axisCommand.anodeMainPnP1AxisX.posAbsolute[2] := #_w1;
END_REGION

REGION Network 88: CmAnodeMainPnP1AxisX Position Absolute Position3
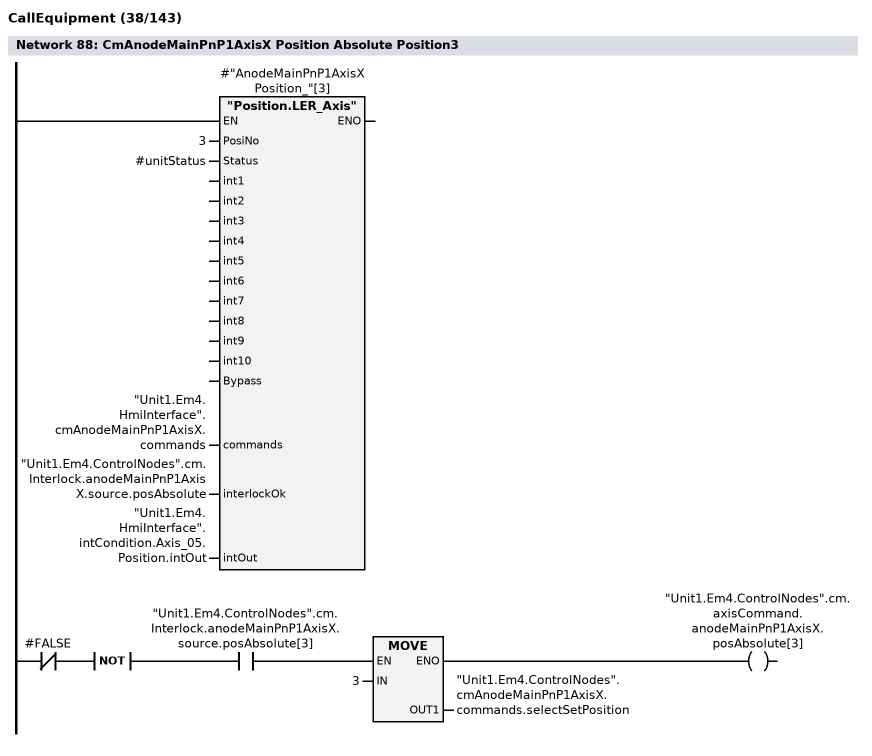
   RUNG wire#powerrail
      #"AnodeMainPnP1AxisX Position_"[3](PosiNo := 3, Status := #unitStatus, int1 :=, int2 :=, int3 :=, int4 :=, int5 :=, int6 :=, int7 :=, int8 :=, int9 :=, int10 :=, Bypass :=, commands := "Unit1.Em4.HmiInterface".cmAnodeMainPnP1AxisX.commands, interlockOk := "Unit1.Em4.ControlNodes".cm.Interlock.anodeMainPnP1AxisX.source.posAbsolute, intOut := "Unit1.Em4.HmiInterface".intCondition.Axis_05.Position.intOut)
   END_RUNG
   RUNG wire#powerrail
      I_Contact( #FALSE )
      Not()
      Contact( "Unit1.Em4.ControlNodes".cm.Interlock.anodeMainPnP1AxisX.source.posAbsolute[3] )
      Move(in := 3, out1 => "Unit1.Em4.ControlNodes".cmAnodeMainPnP1AxisX.commands.selectSetPosition)
      Coil( "Unit1.Em4.ControlNodes".cm.axisCommand.anodeMainPnP1AxisX.posAbsolute[3] )
   END_RUNG
   // the same network as SCL:
   #"AnodeMainPnP1AxisX Position_"[3](PosiNo := 3,   // "Position.LER_Axis"
                           Status := #unitStatus,
                           commands := "Unit1.Em4.HmiInterface".cmAnodeMainPnP1AxisX.commands,
                           interlockOk := "Unit1.Em4.ControlNodes".cm.Interlock.anodeMainPnP1AxisX.source.posAbsolute,
                           intOut := "Unit1.Em4.HmiInterface".intCondition.Axis_05.Position.intOut);
   #_w1 := NOT (NOT #FALSE) AND "Unit1.Em4.ControlNodes".cm.Interlock.anodeMainPnP1AxisX.source.posAbsolute[3];
   IF #_w1 THEN "Unit1.Em4.ControlNodes".cmAnodeMainPnP1AxisX.commands.selectSetPosition := 3; END_IF;
   "Unit1.Em4.ControlNodes".cm.axisCommand.anodeMainPnP1AxisX.posAbsolute[3] := #_w1;
END_REGION

REGION Network 89: CmAnodeMainPnP1AxisX Position Absolute Position4
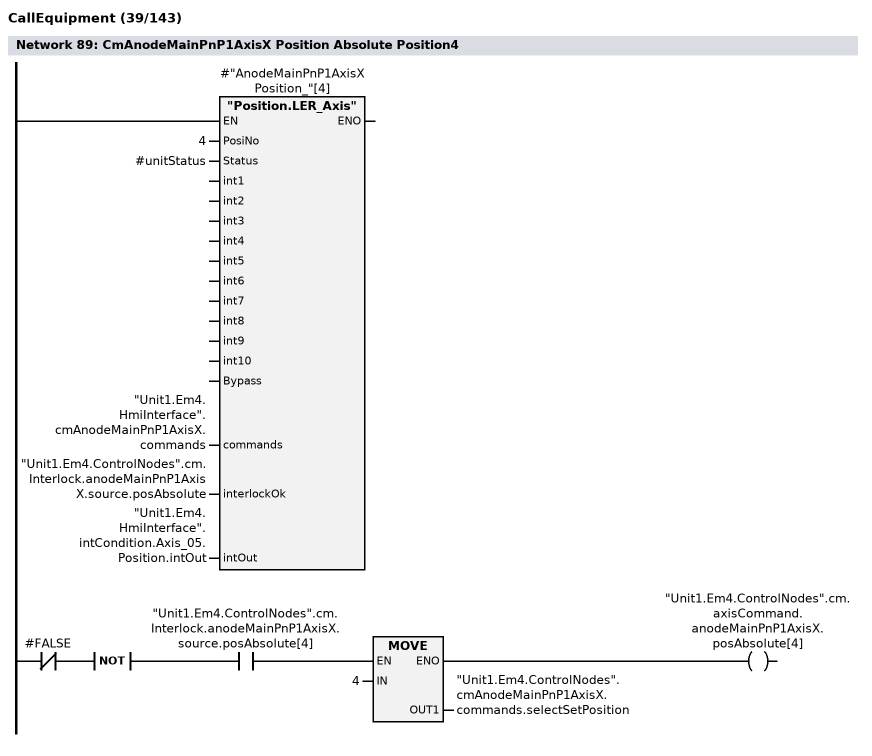
   RUNG wire#powerrail
      #"AnodeMainPnP1AxisX Position_"[4](PosiNo := 4, Status := #unitStatus, int1 :=, int2 :=, int3 :=, int4 :=, int5 :=, int6 :=, int7 :=, int8 :=, int9 :=, int10 :=, Bypass :=, commands := "Unit1.Em4.HmiInterface".cmAnodeMainPnP1AxisX.commands, interlockOk := "Unit1.Em4.ControlNodes".cm.Interlock.anodeMainPnP1AxisX.source.posAbsolute, intOut := "Unit1.Em4.HmiInterface".intCondition.Axis_05.Position.intOut)
   END_RUNG
   RUNG wire#powerrail
      I_Contact( #FALSE )
      Not()
      Contact( "Unit1.Em4.ControlNodes".cm.Interlock.anodeMainPnP1AxisX.source.posAbsolute[4] )
      Move(in := 4, out1 => "Unit1.Em4.ControlNodes".cmAnodeMainPnP1AxisX.commands.selectSetPosition)
      Coil( "Unit1.Em4.ControlNodes".cm.axisCommand.anodeMainPnP1AxisX.posAbsolute[4] )
   END_RUNG
   // the same network as SCL:
   #"AnodeMainPnP1AxisX Position_"[4](PosiNo := 4,   // "Position.LER_Axis"
                           Status := #unitStatus,
                           commands := "Unit1.Em4.HmiInterface".cmAnodeMainPnP1AxisX.commands,
                           interlockOk := "Unit1.Em4.ControlNodes".cm.Interlock.anodeMainPnP1AxisX.source.posAbsolute,
                           intOut := "Unit1.Em4.HmiInterface".intCondition.Axis_05.Position.intOut);
   #_w1 := NOT (NOT #FALSE) AND "Unit1.Em4.ControlNodes".cm.Interlock.anodeMainPnP1AxisX.source.posAbsolute[4];
   IF #_w1 THEN "Unit1.Em4.ControlNodes".cmAnodeMainPnP1AxisX.commands.selectSetPosition := 4; END_IF;
   "Unit1.Em4.ControlNodes".cm.axisCommand.anodeMainPnP1AxisX.posAbsolute[4] := #_w1;
END_REGION

REGION Network 90: CmAnodeMainPnP1AxisX Position Absolute Position5
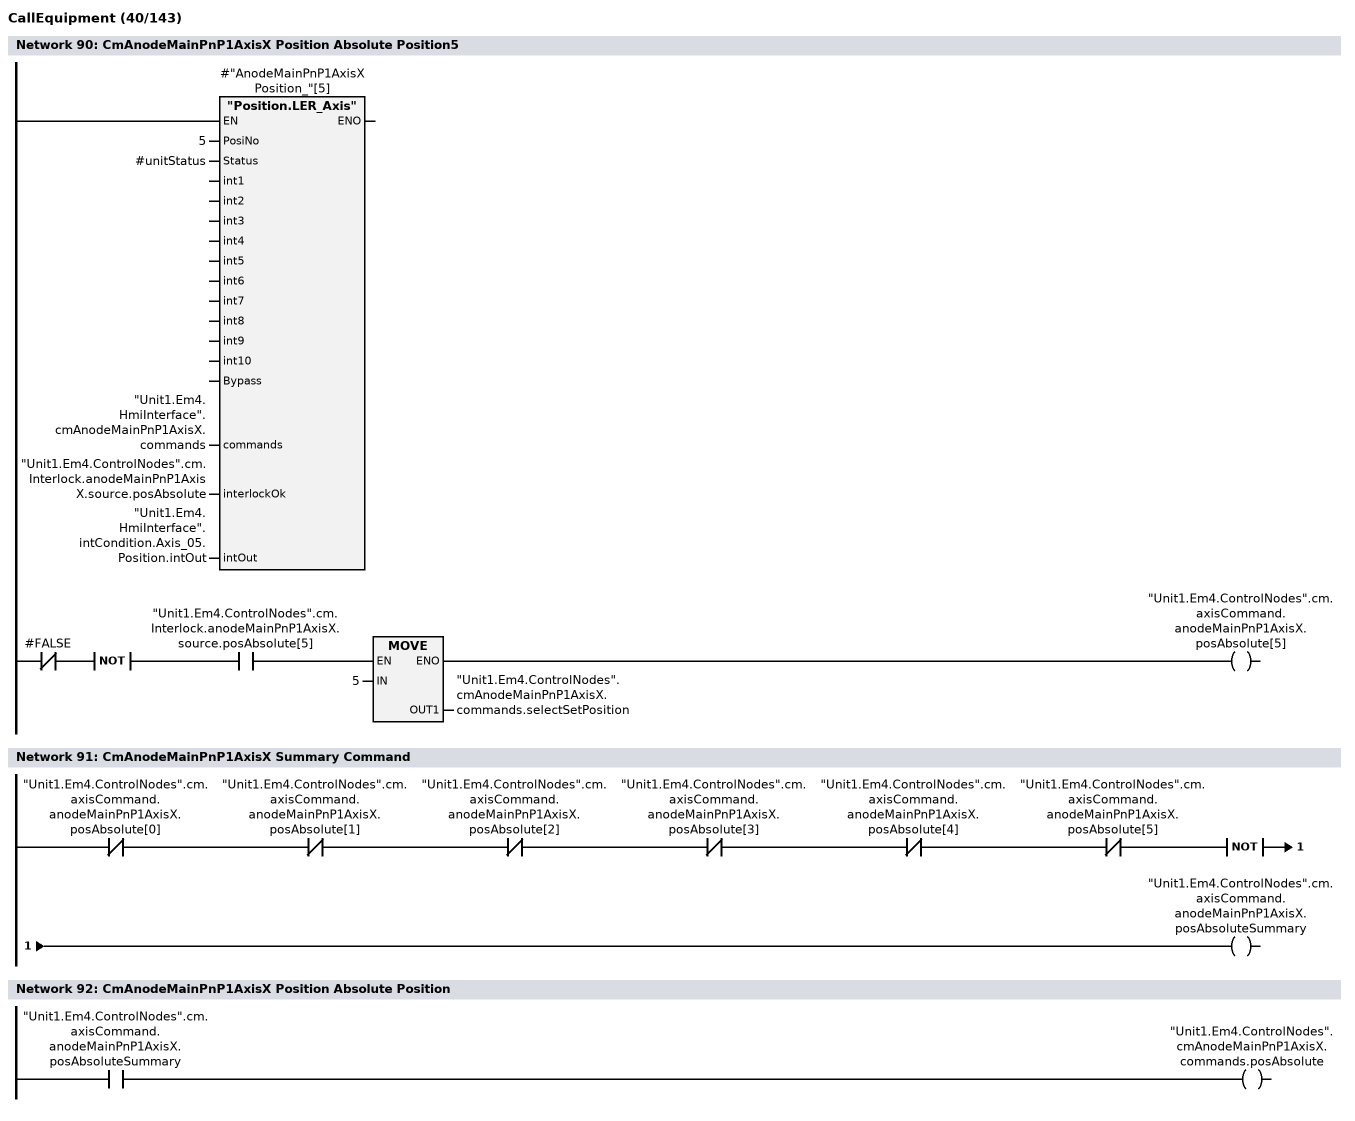
   RUNG wire#powerrail
      #"AnodeMainPnP1AxisX Position_"[5](PosiNo := 5, Status := #unitStatus, int1 :=, int2 :=, int3 :=, int4 :=, int5 :=, int6 :=, int7 :=, int8 :=, int9 :=, int10 :=, Bypass :=, commands := "Unit1.Em4.HmiInterface".cmAnodeMainPnP1AxisX.commands, interlockOk := "Unit1.Em4.ControlNodes".cm.Interlock.anodeMainPnP1AxisX.source.posAbsolute, intOut := "Unit1.Em4.HmiInterface".intCondition.Axis_05.Position.intOut)
   END_RUNG
   RUNG wire#powerrail
      I_Contact( #FALSE )
      Not()
      Contact( "Unit1.Em4.ControlNodes".cm.Interlock.anodeMainPnP1AxisX.source.posAbsolute[5] )
      Move(in := 5, out1 => "Unit1.Em4.ControlNodes".cmAnodeMainPnP1AxisX.commands.selectSetPosition)
      Coil( "Unit1.Em4.ControlNodes".cm.axisCommand.anodeMainPnP1AxisX.posAbsolute[5] )
   END_RUNG
   // the same network as SCL:
   #"AnodeMainPnP1AxisX Position_"[5](PosiNo := 5,   // "Position.LER_Axis"
                           Status := #unitStatus,
                           commands := "Unit1.Em4.HmiInterface".cmAnodeMainPnP1AxisX.commands,
                           interlockOk := "Unit1.Em4.ControlNodes".cm.Interlock.anodeMainPnP1AxisX.source.posAbsolute,
                           intOut := "Unit1.Em4.HmiInterface".intCondition.Axis_05.Position.intOut);
   #_w1 := NOT (NOT #FALSE) AND "Unit1.Em4.ControlNodes".cm.Interlock.anodeMainPnP1AxisX.source.posAbsolute[5];
   IF #_w1 THEN "Unit1.Em4.ControlNodes".cmAnodeMainPnP1AxisX.commands.selectSetPosition := 5; END_IF;
   "Unit1.Em4.ControlNodes".cm.axisCommand.anodeMainPnP1AxisX.posAbsolute[5] := #_w1;
END_REGION

REGION Network 91: CmAnodeMainPnP1AxisX Summary Command
   RUNG wire#powerrail
      I_Contact( "Unit1.Em4.ControlNodes".cm.axisCommand.anodeMainPnP1AxisX.posAbsolute[0] )
      I_Contact( "Unit1.Em4.ControlNodes".cm.axisCommand.anodeMainPnP1AxisX.posAbsolute[1] )
      I_Contact( "Unit1.Em4.ControlNodes".cm.axisCommand.anodeMainPnP1AxisX.posAbsolute[2] )
      I_Contact( "Unit1.Em4.ControlNodes".cm.axisCommand.anodeMainPnP1AxisX.posAbsolute[3] )
      I_Contact( "Unit1.Em4.ControlNodes".cm.axisCommand.anodeMainPnP1AxisX.posAbsolute[4] )
      I_Contact( "Unit1.Em4.ControlNodes".cm.axisCommand.anodeMainPnP1AxisX.posAbsolute[5] )
      Not()
      Coil( "Unit1.Em4.ControlNodes".cm.axisCommand.anodeMainPnP1AxisX.posAbsoluteSummary )
   END_RUNG
   // the same network as SCL:
   "Unit1.Em4.ControlNodes".cm.axisCommand.anodeMainPnP1AxisX.posAbsoluteSummary := NOT (NOT "Unit1.Em4.ControlNodes".cm.axisCommand.anodeMainPnP1AxisX.posAbsolute[0] AND NOT "Unit1.Em4.ControlNodes".cm.axisCommand.anodeMainPnP1AxisX.posAbsolute[1] AND NOT "Unit1.Em4.ControlNodes".cm.axisCommand.anodeMainPnP1AxisX.posAbsolute[2] AND NOT "Unit1.Em4.ControlNodes".cm.axisCommand.anodeMainPnP1AxisX.posAbsolute[3] AND NOT "Unit1.Em4.ControlNodes".cm.axisCommand.anodeMainPnP1AxisX.posAbsolute[4] AND NOT "Unit1.Em4.ControlNodes".cm.axisCommand.anodeMainPnP1AxisX.posAbsolute[5]);
END_REGION

REGION Network 92: CmAnodeMainPnP1AxisX Position Absolute Position
   RUNG wire#powerrail
      Contact( "Unit1.Em4.ControlNodes".cm.axisCommand.anodeMainPnP1AxisX.posAbsoluteSummary )
      Coil( "Unit1.Em4.ControlNodes".cmAnodeMainPnP1AxisX.commands.posAbsolute )
   END_RUNG
   // the same network as SCL:
   "Unit1.Em4.ControlNodes".cmAnodeMainPnP1AxisX.commands.posAbsolute := "Unit1.Em4.ControlNodes".cm.axisCommand.anodeMainPnP1AxisX.posAbsoluteSummary;
END_REGION

REGION Network 93: Call Anode Main P&P 1 X-Axis Interlock Summary
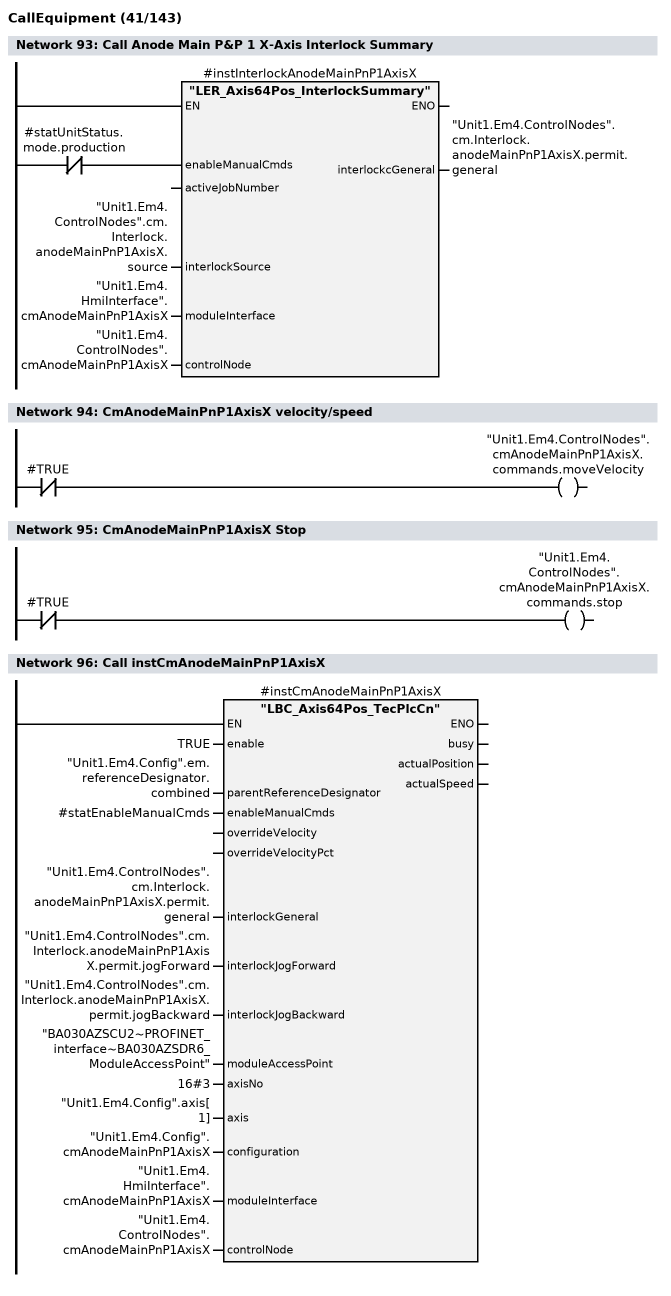
   RUNG wire#powerrail
      #instInterlockAnodeMainPnP1AxisX(enableManualCmds := wire#w1, activeJobNumber :=, interlockSource := "Unit1.Em4.ControlNodes".cm.Interlock.anodeMainPnP1AxisX.source, moduleInterface := "Unit1.Em4.HmiInterface".cmAnodeMainPnP1AxisX, controlNode := "Unit1.Em4.ControlNodes".cmAnodeMainPnP1AxisX, interlockcGeneral => "Unit1.Em4.ControlNodes".cm.Interlock.anodeMainPnP1AxisX.permit.general)
   END_RUNG
   RUNG wire#powerrail
      I_Contact( #statUnitStatus.mode.production )
   END_RUNG wire#w1
   // the same network as SCL:
   #instInterlockAnodeMainPnP1AxisX(enableManualCmds := NOT #statUnitStatus.mode.production,   // "LER_Axis64Pos_InterlockSummary"
                           interlockSource := "Unit1.Em4.ControlNodes".cm.Interlock.anodeMainPnP1AxisX.source,
                           moduleInterface := "Unit1.Em4.HmiInterface".cmAnodeMainPnP1AxisX,
                           controlNode := "Unit1.Em4.ControlNodes".cmAnodeMainPnP1AxisX,
                           interlockcGeneral => "Unit1.Em4.ControlNodes".cm.Interlock.anodeMainPnP1AxisX.permit.general);
END_REGION

REGION Network 94: CmAnodeMainPnP1AxisX velocity/speed
   RUNG wire#powerrail
      I_Contact( #TRUE )
      Coil( "Unit1.Em4.ControlNodes".cmAnodeMainPnP1AxisX.commands.moveVelocity )
   END_RUNG
   // the same network as SCL:
   "Unit1.Em4.ControlNodes".cmAnodeMainPnP1AxisX.commands.moveVelocity := NOT #TRUE;
END_REGION

REGION Network 95: CmAnodeMainPnP1AxisX Stop
   RUNG wire#powerrail
      I_Contact( #TRUE )
      Coil( "Unit1.Em4.ControlNodes".cmAnodeMainPnP1AxisX.commands.stop )
   END_RUNG
   // the same network as SCL:
   "Unit1.Em4.ControlNodes".cmAnodeMainPnP1AxisX.commands.stop := NOT #TRUE;
END_REGION

REGION Network 96: Call instCmAnodeMainPnP1AxisX
   RUNG wire#powerrail
      #instCmAnodeMainPnP1AxisX(enable := TRUE, parentReferenceDesignator := "Unit1.Em4.Config".em.referenceDesignator.combined, enableManualCmds := #statEnableManualCmds, overrideVelocity :=, overrideVelocityPct :=, interlockGeneral := "Unit1.Em4.ControlNodes".cm.Interlock.anodeMainPnP1AxisX.permit.general, interlockJogForward := "Unit1.Em4.ControlNodes".cm.Interlock.anodeMainPnP1AxisX.permit.jogForward, interlockJogBackward := "Unit1.Em4.ControlNodes".cm.Interlock.anodeMainPnP1AxisX.permit.jogBackward, moduleAccessPoint := "BA030AZSCU2~PROFINET_interface~BA030AZSDR6_ModuleAccessPoint", axisNo := 16#3, axis := "Unit1.Em4.Config".axis[1], configuration := "Unit1.Em4.Config".cmAnodeMainPnP1AxisX, moduleInterface := "Unit1.Em4.HmiInterface".cmAnodeMainPnP1AxisX, controlNode := "Unit1.Em4.ControlNodes".cmAnodeMainPnP1AxisX, busy =>, actualPosition =>, actualSpeed =>)
   END_RUNG
   // the same network as SCL:
   #instCmAnodeMainPnP1AxisX(enable := TRUE,   // "LBC_Axis64Pos_TecPlcCn"
                           parentReferenceDesignator := "Unit1.Em4.Config".em.referenceDesignator.combined,
                           enableManualCmds := #statEnableManualCmds,
                           interlockGeneral := "Unit1.Em4.ControlNodes".cm.Interlock.anodeMainPnP1AxisX.permit.general,
                           interlockJogForward := "Unit1.Em4.ControlNodes".cm.Interlock.anodeMainPnP1AxisX.permit.jogForward,
                           interlockJogBackward := "Unit1.Em4.ControlNodes".cm.Interlock.anodeMainPnP1AxisX.permit.jogBackward,
                           moduleAccessPoint := "BA030AZSCU2~PROFINET_interface~BA030AZSDR6_ModuleAccessPoint",
                           axisNo := 16#3,
                           axis := "Unit1.Em4.Config".axis[1],
                           configuration := "Unit1.Em4.Config".cmAnodeMainPnP1AxisX,
                           moduleInterface := "Unit1.Em4.HmiInterface".cmAnodeMainPnP1AxisX,
                           controlNode := "Unit1.Em4.ControlNodes".cmAnodeMainPnP1AxisX);
END_REGION

REGION Network 97: CmAnodeMainPnP1AxisX SoftCam
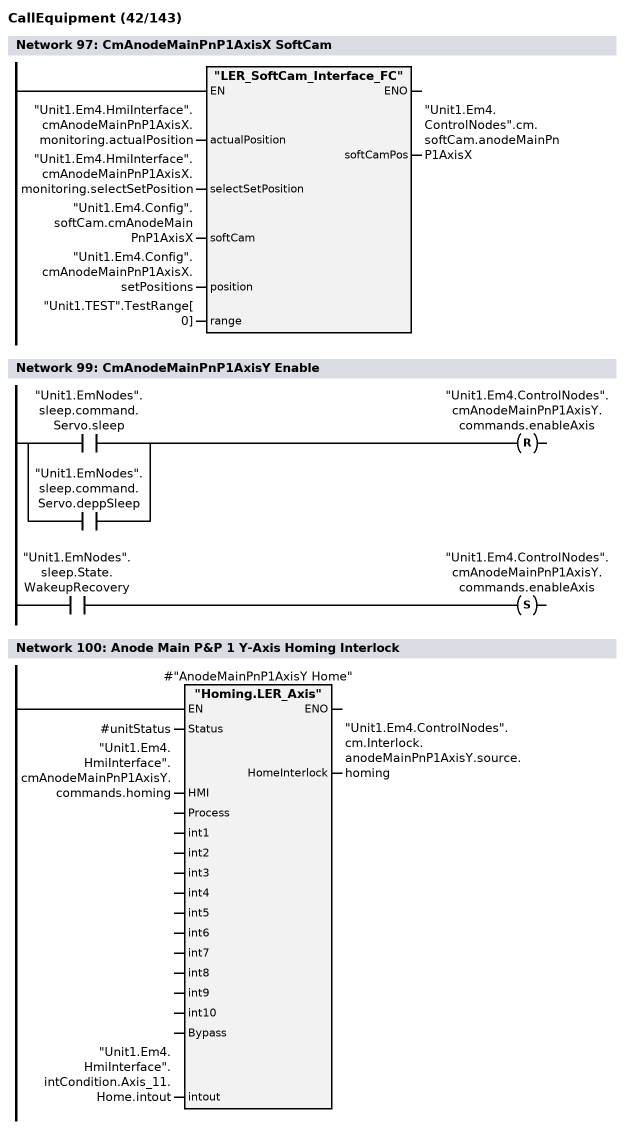
   RUNG wire#powerrail
      "LER_SoftCam_Interface_FC"(actualPosition := "Unit1.Em4.HmiInterface".cmAnodeMainPnP1AxisX.monitoring.actualPosition, selectSetPosition := "Unit1.Em4.HmiInterface".cmAnodeMainPnP1AxisX.monitoring.selectSetPosition, softCam := "Unit1.Em4.Config".softCam.cmAnodeMainPnP1AxisX, position := "Unit1.Em4.Config".cmAnodeMainPnP1AxisX.setPositions, range := "Unit1.TEST".TestRange[0], softCamPos => "Unit1.Em4.ControlNodes".cm.softCam.anodeMainPnP1AxisX)
   END_RUNG
   // the same network as SCL:
   "LER_SoftCam_Interface_FC"(actualPosition := "Unit1.Em4.HmiInterface".cmAnodeMainPnP1AxisX.monitoring.actualPosition,
                           selectSetPosition := "Unit1.Em4.HmiInterface".cmAnodeMainPnP1AxisX.monitoring.selectSetPosition,
                           softCam := "Unit1.Em4.Config".softCam.cmAnodeMainPnP1AxisX,
                           position := "Unit1.Em4.Config".cmAnodeMainPnP1AxisX.setPositions,
                           range := "Unit1.TEST".TestRange[0],
                           softCamPos => "Unit1.Em4.ControlNodes".cm.softCam.anodeMainPnP1AxisX);
END_REGION

REGION Network 99: CmAnodeMainPnP1AxisY Enable
   RUNG wire#powerrail
      Contact( "Unit1.EmNodes".sleep.command.Servo.sleep )
      wire#w1
      R_Coil( "Unit1.Em4.ControlNodes".cmAnodeMainPnP1AxisY.commands.enableAxis )
   END_RUNG
   RUNG wire#powerrail
      Contact( "Unit1.EmNodes".sleep.command.Servo.deppSleep )
   END_RUNG wire#w1
   RUNG wire#powerrail
      Contact( "Unit1.EmNodes".sleep.State.WakeupRecovery )
      S_Coil( "Unit1.Em4.ControlNodes".cmAnodeMainPnP1AxisY.commands.enableAxis )
   END_RUNG
   // the same network as SCL:
   IF "Unit1.EmNodes".sleep.command.Servo.sleep OR "Unit1.EmNodes".sleep.command.Servo.deppSleep THEN
       "Unit1.Em4.ControlNodes".cmAnodeMainPnP1AxisY.commands.enableAxis := FALSE;
   END_IF;
   IF "Unit1.EmNodes".sleep.State.WakeupRecovery THEN
       "Unit1.Em4.ControlNodes".cmAnodeMainPnP1AxisY.commands.enableAxis := TRUE;
   END_IF;
END_REGION

REGION Network 100: Anode Main P&P 1 Y-Axis Homing Interlock
   RUNG wire#powerrail
      #"AnodeMainPnP1AxisY Home"(Status := #unitStatus, HMI := "Unit1.Em4.HmiInterface".cmAnodeMainPnP1AxisY.commands.homing, Process :=, int1 :=, int2 :=, int3 :=, int4 :=, int5 :=, int6 :=, int7 :=, int8 :=, int9 :=, int10 :=, Bypass :=, intout := "Unit1.Em4.HmiInterface".intCondition.Axis_11.Home.intout, HomeInterlock => "Unit1.Em4.ControlNodes".cm.Interlock.anodeMainPnP1AxisY.source.homing)
   END_RUNG
   // the same network as SCL:
   #"AnodeMainPnP1AxisY Home"(Status := #unitStatus,   // "Homing.LER_Axis"
                           HMI := "Unit1.Em4.HmiInterface".cmAnodeMainPnP1AxisY.commands.homing,
                           intout := "Unit1.Em4.HmiInterface".intCondition.Axis_11.Home.intout,
                           HomeInterlock => "Unit1.Em4.ControlNodes".cm.Interlock.anodeMainPnP1AxisY.source.homing);
END_REGION

REGION Network 101: CmAnodeMainPnP1AxisY Position Absolute Jog
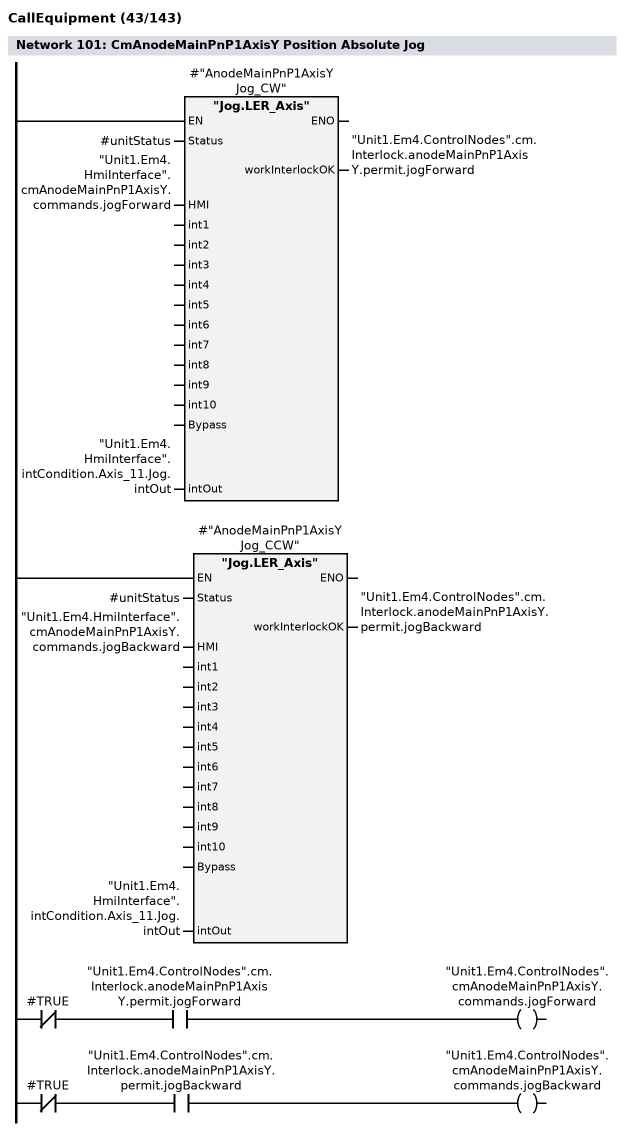
   RUNG wire#powerrail
      #"AnodeMainPnP1AxisY Jog_CW"(Status := #unitStatus, HMI := "Unit1.Em4.HmiInterface".cmAnodeMainPnP1AxisY.commands.jogForward, int1 :=, int2 :=, int3 :=, int4 :=, int5 :=, int6 :=, int7 :=, int8 :=, int9 :=, int10 :=, Bypass :=, intOut := "Unit1.Em4.HmiInterface".intCondition.Axis_11.Jog.intOut, workInterlockOK => "Unit1.Em4.ControlNodes".cm.Interlock.anodeMainPnP1AxisY.permit.jogForward)
   END_RUNG
   RUNG wire#powerrail
      #"AnodeMainPnP1AxisY Jog_CCW"(Status := #unitStatus, HMI := "Unit1.Em4.HmiInterface".cmAnodeMainPnP1AxisY.commands.jogBackward, int1 :=, int2 :=, int3 :=, int4 :=, int5 :=, int6 :=, int7 :=, int8 :=, int9 :=, int10 :=, Bypass :=, intOut := "Unit1.Em4.HmiInterface".intCondition.Axis_11.Jog.intOut, workInterlockOK => "Unit1.Em4.ControlNodes".cm.Interlock.anodeMainPnP1AxisY.permit.jogBackward)
   END_RUNG
   RUNG wire#powerrail
      I_Contact( #TRUE )
      Contact( "Unit1.Em4.ControlNodes".cm.Interlock.anodeMainPnP1AxisY.permit.jogForward )
      Coil( "Unit1.Em4.ControlNodes".cmAnodeMainPnP1AxisY.commands.jogForward )
   END_RUNG
   RUNG wire#powerrail
      I_Contact( #TRUE )
      Contact( "Unit1.Em4.ControlNodes".cm.Interlock.anodeMainPnP1AxisY.permit.jogBackward )
      Coil( "Unit1.Em4.ControlNodes".cmAnodeMainPnP1AxisY.commands.jogBackward )
   END_RUNG
   // the same network as SCL:
   #"AnodeMainPnP1AxisY Jog_CW"(Status := #unitStatus,   // "Jog.LER_Axis"
                           HMI := "Unit1.Em4.HmiInterface".cmAnodeMainPnP1AxisY.commands.jogForward,
                           intOut := "Unit1.Em4.HmiInterface".intCondition.Axis_11.Jog.intOut,
                           workInterlockOK => "Unit1.Em4.ControlNodes".cm.Interlock.anodeMainPnP1AxisY.permit.jogForward);
   #"AnodeMainPnP1AxisY Jog_CCW"(Status := #unitStatus,   // "Jog.LER_Axis"
                           HMI := "Unit1.Em4.HmiInterface".cmAnodeMainPnP1AxisY.commands.jogBackward,
                           intOut := "Unit1.Em4.HmiInterface".intCondition.Axis_11.Jog.intOut,
                           workInterlockOK => "Unit1.Em4.ControlNodes".cm.Interlock.anodeMainPnP1AxisY.permit.jogBackward);
   "Unit1.Em4.ControlNodes".cmAnodeMainPnP1AxisY.commands.jogForward := NOT #TRUE AND "Unit1.Em4.ControlNodes".cm.Interlock.anodeMainPnP1AxisY.permit.jogForward;
   "Unit1.Em4.ControlNodes".cmAnodeMainPnP1AxisY.commands.jogBackward := NOT #TRUE AND "Unit1.Em4.ControlNodes".cm.Interlock.anodeMainPnP1AxisY.permit.jogBackward;
END_REGION

REGION Network 102: CmAnodeMainPnP1AxisY Position Absolute Position0
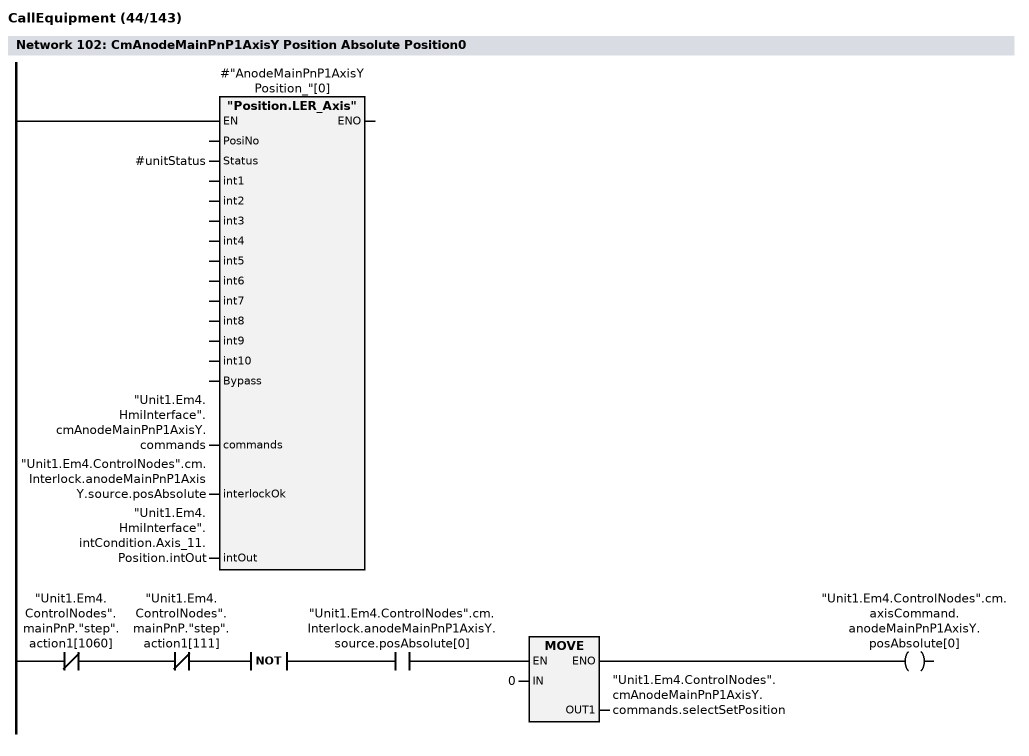
   RUNG wire#powerrail
      #"AnodeMainPnP1AxisY Position_"[0](PosiNo :=, Status := #unitStatus, int1 :=, int2 :=, int3 :=, int4 :=, int5 :=, int6 :=, int7 :=, int8 :=, int9 :=, int10 :=, Bypass :=, commands := "Unit1.Em4.HmiInterface".cmAnodeMainPnP1AxisY.commands, interlockOk := "Unit1.Em4.ControlNodes".cm.Interlock.anodeMainPnP1AxisY.source.posAbsolute, intOut := "Unit1.Em4.HmiInterface".intCondition.Axis_11.Position.intOut)
   END_RUNG
   RUNG wire#powerrail
      I_Contact( "Unit1.Em4.ControlNodes".mainPnP."step".action1[1060] )
      I_Contact( "Unit1.Em4.ControlNodes".mainPnP."step".action1[111] )
      Not()
      Contact( "Unit1.Em4.ControlNodes".cm.Interlock.anodeMainPnP1AxisY.source.posAbsolute[0] )
      Move(in := 0, out1 => "Unit1.Em4.ControlNodes".cmAnodeMainPnP1AxisY.commands.selectSetPosition)
      Coil( "Unit1.Em4.ControlNodes".cm.axisCommand.anodeMainPnP1AxisY.posAbsolute[0] )
   END_RUNG
   // the same network as SCL:
   #"AnodeMainPnP1AxisY Position_"[0](Status := #unitStatus,   // "Position.LER_Axis"
                           commands := "Unit1.Em4.HmiInterface".cmAnodeMainPnP1AxisY.commands,
                           interlockOk := "Unit1.Em4.ControlNodes".cm.Interlock.anodeMainPnP1AxisY.source.posAbsolute,
                           intOut := "Unit1.Em4.HmiInterface".intCondition.Axis_11.Position.intOut);
   #_w1 := NOT (NOT "Unit1.Em4.ControlNodes".mainPnP."step".action1[1060] AND NOT "Unit1.Em4.ControlNodes".mainPnP."step".action1[111]) AND "Unit1.Em4.ControlNodes".cm.Interlock.anodeMainPnP1AxisY.source.posAbsolute[0];
   IF #_w1 THEN "Unit1.Em4.ControlNodes".cmAnodeMainPnP1AxisY.commands.selectSetPosition := 0; END_IF;
   "Unit1.Em4.ControlNodes".cm.axisCommand.anodeMainPnP1AxisY.posAbsolute[0] := #_w1;
END_REGION

REGION Network 103: CmAnodeMainPnP1AxisY Position Absolute Position1
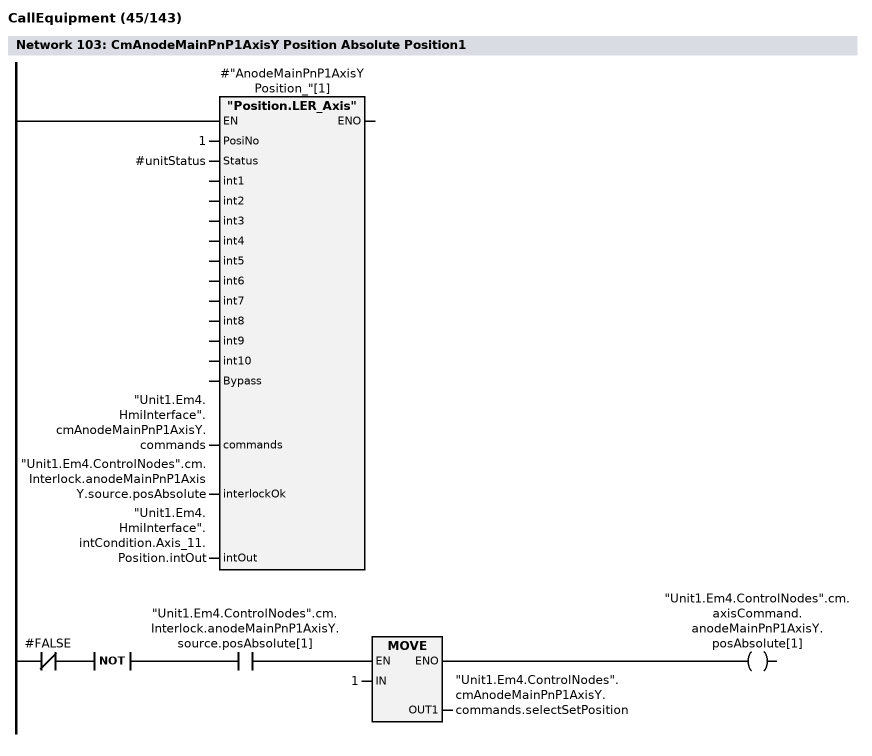
   RUNG wire#powerrail
      #"AnodeMainPnP1AxisY Position_"[1](PosiNo := 1, Status := #unitStatus, int1 :=, int2 :=, int3 :=, int4 :=, int5 :=, int6 :=, int7 :=, int8 :=, int9 :=, int10 :=, Bypass :=, commands := "Unit1.Em4.HmiInterface".cmAnodeMainPnP1AxisY.commands, interlockOk := "Unit1.Em4.ControlNodes".cm.Interlock.anodeMainPnP1AxisY.source.posAbsolute, intOut := "Unit1.Em4.HmiInterface".intCondition.Axis_11.Position.intOut)
   END_RUNG
   RUNG wire#powerrail
      I_Contact( #FALSE )
      Not()
      Contact( "Unit1.Em4.ControlNodes".cm.Interlock.anodeMainPnP1AxisY.source.posAbsolute[1] )
      Move(in := 1, out1 => "Unit1.Em4.ControlNodes".cmAnodeMainPnP1AxisY.commands.selectSetPosition)
      Coil( "Unit1.Em4.ControlNodes".cm.axisCommand.anodeMainPnP1AxisY.posAbsolute[1] )
   END_RUNG
   // the same network as SCL:
   #"AnodeMainPnP1AxisY Position_"[1](PosiNo := 1,   // "Position.LER_Axis"
                           Status := #unitStatus,
                           commands := "Unit1.Em4.HmiInterface".cmAnodeMainPnP1AxisY.commands,
                           interlockOk := "Unit1.Em4.ControlNodes".cm.Interlock.anodeMainPnP1AxisY.source.posAbsolute,
                           intOut := "Unit1.Em4.HmiInterface".intCondition.Axis_11.Position.intOut);
   #_w1 := NOT (NOT #FALSE) AND "Unit1.Em4.ControlNodes".cm.Interlock.anodeMainPnP1AxisY.source.posAbsolute[1];
   IF #_w1 THEN "Unit1.Em4.ControlNodes".cmAnodeMainPnP1AxisY.commands.selectSetPosition := 1; END_IF;
   "Unit1.Em4.ControlNodes".cm.axisCommand.anodeMainPnP1AxisY.posAbsolute[1] := #_w1;
END_REGION

REGION Network 104: CmAnodeMainPnP1AxisY Position Absolute Position2
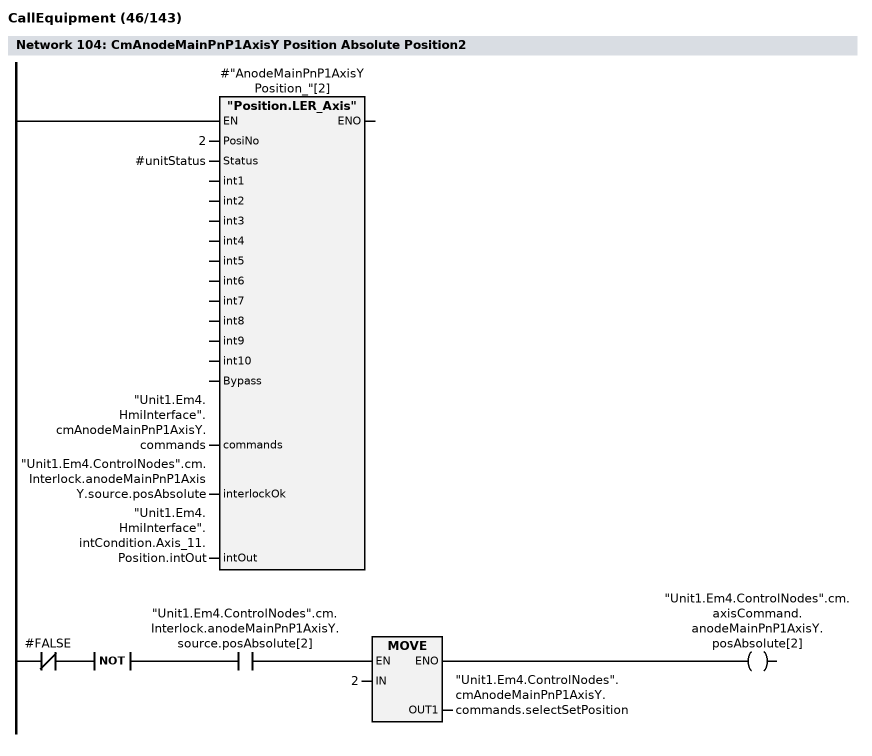
   RUNG wire#powerrail
      #"AnodeMainPnP1AxisY Position_"[2](PosiNo := 2, Status := #unitStatus, int1 :=, int2 :=, int3 :=, int4 :=, int5 :=, int6 :=, int7 :=, int8 :=, int9 :=, int10 :=, Bypass :=, commands := "Unit1.Em4.HmiInterface".cmAnodeMainPnP1AxisY.commands, interlockOk := "Unit1.Em4.ControlNodes".cm.Interlock.anodeMainPnP1AxisY.source.posAbsolute, intOut := "Unit1.Em4.HmiInterface".intCondition.Axis_11.Position.intOut)
   END_RUNG
   RUNG wire#powerrail
      I_Contact( #FALSE )
      Not()
      Contact( "Unit1.Em4.ControlNodes".cm.Interlock.anodeMainPnP1AxisY.source.posAbsolute[2] )
      Move(in := 2, out1 => "Unit1.Em4.ControlNodes".cmAnodeMainPnP1AxisY.commands.selectSetPosition)
      Coil( "Unit1.Em4.ControlNodes".cm.axisCommand.anodeMainPnP1AxisY.posAbsolute[2] )
   END_RUNG
   // the same network as SCL:
   #"AnodeMainPnP1AxisY Position_"[2](PosiNo := 2,   // "Position.LER_Axis"
                           Status := #unitStatus,
                           commands := "Unit1.Em4.HmiInterface".cmAnodeMainPnP1AxisY.commands,
                           interlockOk := "Unit1.Em4.ControlNodes".cm.Interlock.anodeMainPnP1AxisY.source.posAbsolute,
                           intOut := "Unit1.Em4.HmiInterface".intCondition.Axis_11.Position.intOut);
   #_w1 := NOT (NOT #FALSE) AND "Unit1.Em4.ControlNodes".cm.Interlock.anodeMainPnP1AxisY.source.posAbsolute[2];
   IF #_w1 THEN "Unit1.Em4.ControlNodes".cmAnodeMainPnP1AxisY.commands.selectSetPosition := 2; END_IF;
   "Unit1.Em4.ControlNodes".cm.axisCommand.anodeMainPnP1AxisY.posAbsolute[2] := #_w1;
END_REGION

REGION Network 105: CmAnodeMainPnP1AxisY Position Absolute Position3
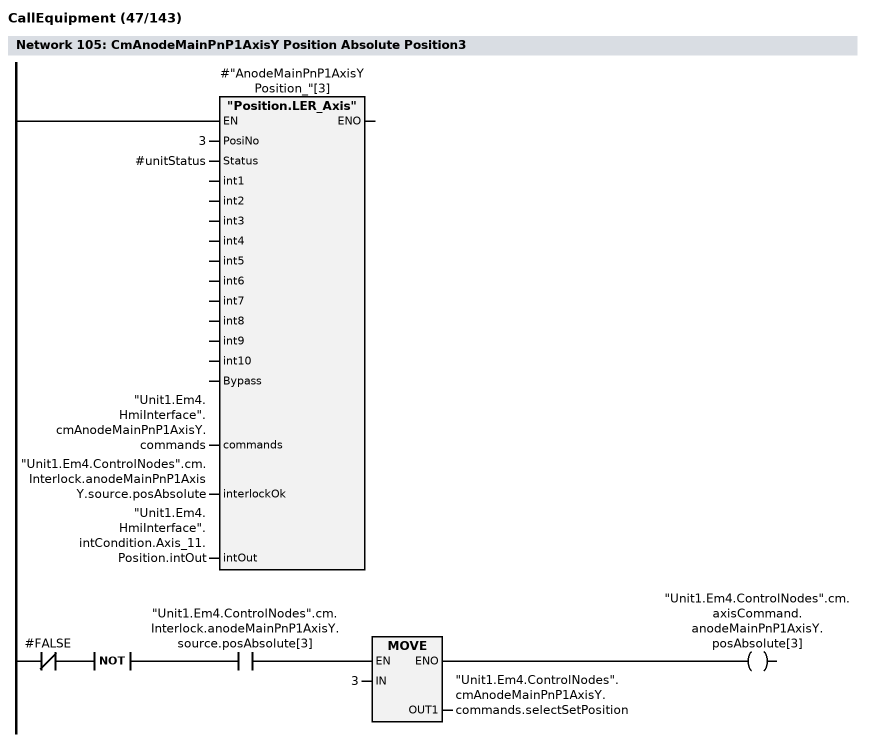
   RUNG wire#powerrail
      #"AnodeMainPnP1AxisY Position_"[3](PosiNo := 3, Status := #unitStatus, int1 :=, int2 :=, int3 :=, int4 :=, int5 :=, int6 :=, int7 :=, int8 :=, int9 :=, int10 :=, Bypass :=, commands := "Unit1.Em4.HmiInterface".cmAnodeMainPnP1AxisY.commands, interlockOk := "Unit1.Em4.ControlNodes".cm.Interlock.anodeMainPnP1AxisY.source.posAbsolute, intOut := "Unit1.Em4.HmiInterface".intCondition.Axis_11.Position.intOut)
   END_RUNG
   RUNG wire#powerrail
      I_Contact( #FALSE )
      Not()
      Contact( "Unit1.Em4.ControlNodes".cm.Interlock.anodeMainPnP1AxisY.source.posAbsolute[3] )
      Move(in := 3, out1 => "Unit1.Em4.ControlNodes".cmAnodeMainPnP1AxisY.commands.selectSetPosition)
      Coil( "Unit1.Em4.ControlNodes".cm.axisCommand.anodeMainPnP1AxisY.posAbsolute[3] )
   END_RUNG
   // the same network as SCL:
   #"AnodeMainPnP1AxisY Position_"[3](PosiNo := 3,   // "Position.LER_Axis"
                           Status := #unitStatus,
                           commands := "Unit1.Em4.HmiInterface".cmAnodeMainPnP1AxisY.commands,
                           interlockOk := "Unit1.Em4.ControlNodes".cm.Interlock.anodeMainPnP1AxisY.source.posAbsolute,
                           intOut := "Unit1.Em4.HmiInterface".intCondition.Axis_11.Position.intOut);
   #_w1 := NOT (NOT #FALSE) AND "Unit1.Em4.ControlNodes".cm.Interlock.anodeMainPnP1AxisY.source.posAbsolute[3];
   IF #_w1 THEN "Unit1.Em4.ControlNodes".cmAnodeMainPnP1AxisY.commands.selectSetPosition := 3; END_IF;
   "Unit1.Em4.ControlNodes".cm.axisCommand.anodeMainPnP1AxisY.posAbsolute[3] := #_w1;
END_REGION

REGION Network 106: CmAnodeMainPnP1AxisY Position Absolute Position4
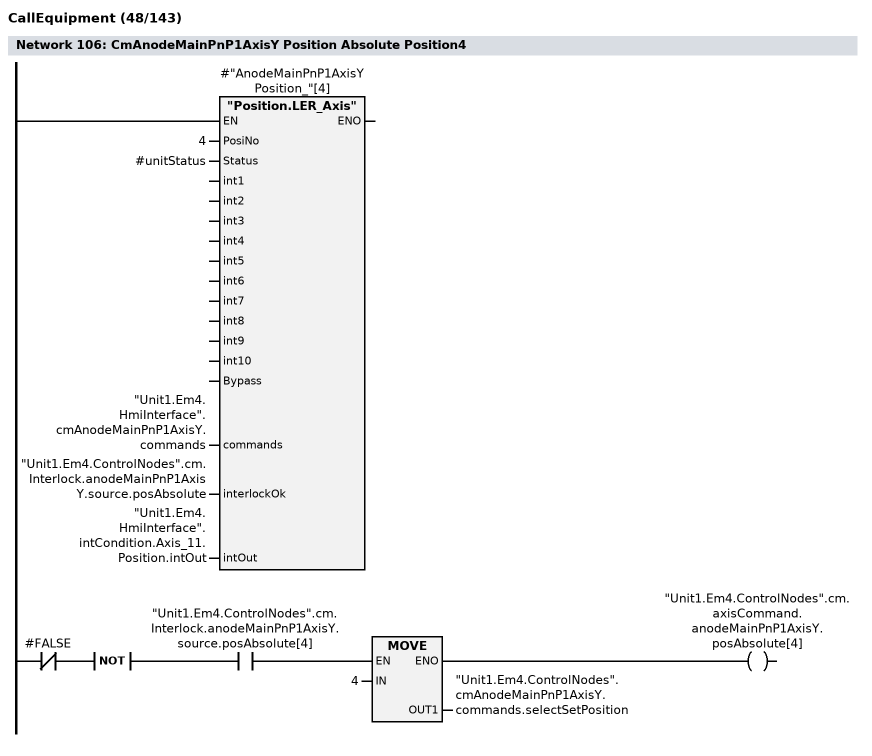
   RUNG wire#powerrail
      #"AnodeMainPnP1AxisY Position_"[4](PosiNo := 4, Status := #unitStatus, int1 :=, int2 :=, int3 :=, int4 :=, int5 :=, int6 :=, int7 :=, int8 :=, int9 :=, int10 :=, Bypass :=, commands := "Unit1.Em4.HmiInterface".cmAnodeMainPnP1AxisY.commands, interlockOk := "Unit1.Em4.ControlNodes".cm.Interlock.anodeMainPnP1AxisY.source.posAbsolute, intOut := "Unit1.Em4.HmiInterface".intCondition.Axis_11.Position.intOut)
   END_RUNG
   RUNG wire#powerrail
      I_Contact( #FALSE )
      Not()
      Contact( "Unit1.Em4.ControlNodes".cm.Interlock.anodeMainPnP1AxisY.source.posAbsolute[4] )
      Move(in := 4, out1 => "Unit1.Em4.ControlNodes".cmAnodeMainPnP1AxisY.commands.selectSetPosition)
      Coil( "Unit1.Em4.ControlNodes".cm.axisCommand.anodeMainPnP1AxisY.posAbsolute[4] )
   END_RUNG
   // the same network as SCL:
   #"AnodeMainPnP1AxisY Position_"[4](PosiNo := 4,   // "Position.LER_Axis"
                           Status := #unitStatus,
                           commands := "Unit1.Em4.HmiInterface".cmAnodeMainPnP1AxisY.commands,
                           interlockOk := "Unit1.Em4.ControlNodes".cm.Interlock.anodeMainPnP1AxisY.source.posAbsolute,
                           intOut := "Unit1.Em4.HmiInterface".intCondition.Axis_11.Position.intOut);
   #_w1 := NOT (NOT #FALSE) AND "Unit1.Em4.ControlNodes".cm.Interlock.anodeMainPnP1AxisY.source.posAbsolute[4];
   IF #_w1 THEN "Unit1.Em4.ControlNodes".cmAnodeMainPnP1AxisY.commands.selectSetPosition := 4; END_IF;
   "Unit1.Em4.ControlNodes".cm.axisCommand.anodeMainPnP1AxisY.posAbsolute[4] := #_w1;
END_REGION

REGION Network 107: CmAnodeMainPnP1AxisY Position Absolute Position5
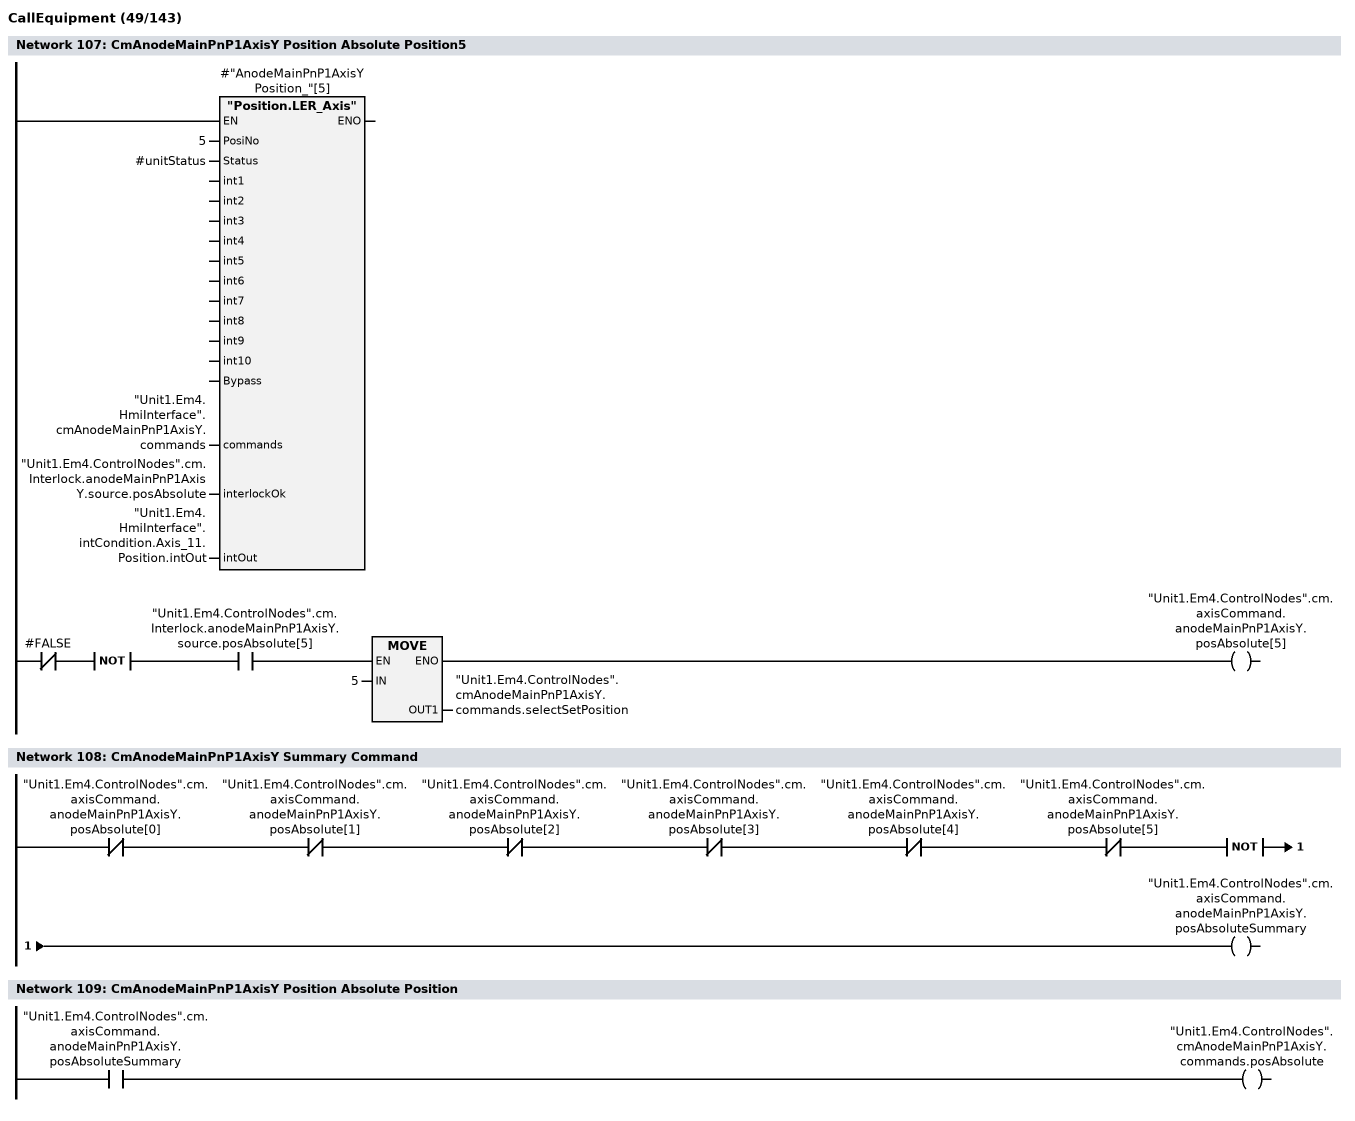
   RUNG wire#powerrail
      #"AnodeMainPnP1AxisY Position_"[5](PosiNo := 5, Status := #unitStatus, int1 :=, int2 :=, int3 :=, int4 :=, int5 :=, int6 :=, int7 :=, int8 :=, int9 :=, int10 :=, Bypass :=, commands := "Unit1.Em4.HmiInterface".cmAnodeMainPnP1AxisY.commands, interlockOk := "Unit1.Em4.ControlNodes".cm.Interlock.anodeMainPnP1AxisY.source.posAbsolute, intOut := "Unit1.Em4.HmiInterface".intCondition.Axis_11.Position.intOut)
   END_RUNG
   RUNG wire#powerrail
      I_Contact( #FALSE )
      Not()
      Contact( "Unit1.Em4.ControlNodes".cm.Interlock.anodeMainPnP1AxisY.source.posAbsolute[5] )
      Move(in := 5, out1 => "Unit1.Em4.ControlNodes".cmAnodeMainPnP1AxisY.commands.selectSetPosition)
      Coil( "Unit1.Em4.ControlNodes".cm.axisCommand.anodeMainPnP1AxisY.posAbsolute[5] )
   END_RUNG
   // the same network as SCL:
   #"AnodeMainPnP1AxisY Position_"[5](PosiNo := 5,   // "Position.LER_Axis"
                           Status := #unitStatus,
                           commands := "Unit1.Em4.HmiInterface".cmAnodeMainPnP1AxisY.commands,
                           interlockOk := "Unit1.Em4.ControlNodes".cm.Interlock.anodeMainPnP1AxisY.source.posAbsolute,
                           intOut := "Unit1.Em4.HmiInterface".intCondition.Axis_11.Position.intOut);
   #_w1 := NOT (NOT #FALSE) AND "Unit1.Em4.ControlNodes".cm.Interlock.anodeMainPnP1AxisY.source.posAbsolute[5];
   IF #_w1 THEN "Unit1.Em4.ControlNodes".cmAnodeMainPnP1AxisY.commands.selectSetPosition := 5; END_IF;
   "Unit1.Em4.ControlNodes".cm.axisCommand.anodeMainPnP1AxisY.posAbsolute[5] := #_w1;
END_REGION

REGION Network 108: CmAnodeMainPnP1AxisY Summary Command
   RUNG wire#powerrail
      I_Contact( "Unit1.Em4.ControlNodes".cm.axisCommand.anodeMainPnP1AxisY.posAbsolute[0] )
      I_Contact( "Unit1.Em4.ControlNodes".cm.axisCommand.anodeMainPnP1AxisY.posAbsolute[1] )
      I_Contact( "Unit1.Em4.ControlNodes".cm.axisCommand.anodeMainPnP1AxisY.posAbsolute[2] )
      I_Contact( "Unit1.Em4.ControlNodes".cm.axisCommand.anodeMainPnP1AxisY.posAbsolute[3] )
      I_Contact( "Unit1.Em4.ControlNodes".cm.axisCommand.anodeMainPnP1AxisY.posAbsolute[4] )
      I_Contact( "Unit1.Em4.ControlNodes".cm.axisCommand.anodeMainPnP1AxisY.posAbsolute[5] )
      Not()
      Coil( "Unit1.Em4.ControlNodes".cm.axisCommand.anodeMainPnP1AxisY.posAbsoluteSummary )
   END_RUNG
   // the same network as SCL:
   "Unit1.Em4.ControlNodes".cm.axisCommand.anodeMainPnP1AxisY.posAbsoluteSummary := NOT (NOT "Unit1.Em4.ControlNodes".cm.axisCommand.anodeMainPnP1AxisY.posAbsolute[0] AND NOT "Unit1.Em4.ControlNodes".cm.axisCommand.anodeMainPnP1AxisY.posAbsolute[1] AND NOT "Unit1.Em4.ControlNodes".cm.axisCommand.anodeMainPnP1AxisY.posAbsolute[2] AND NOT "Unit1.Em4.ControlNodes".cm.axisCommand.anodeMainPnP1AxisY.posAbsolute[3] AND NOT "Unit1.Em4.ControlNodes".cm.axisCommand.anodeMainPnP1AxisY.posAbsolute[4] AND NOT "Unit1.Em4.ControlNodes".cm.axisCommand.anodeMainPnP1AxisY.posAbsolute[5]);
END_REGION

REGION Network 109: CmAnodeMainPnP1AxisY Position Absolute Position
   RUNG wire#powerrail
      Contact( "Unit1.Em4.ControlNodes".cm.axisCommand.anodeMainPnP1AxisY.posAbsoluteSummary )
      Coil( "Unit1.Em4.ControlNodes".cmAnodeMainPnP1AxisY.commands.posAbsolute )
   END_RUNG
   // the same network as SCL:
   "Unit1.Em4.ControlNodes".cmAnodeMainPnP1AxisY.commands.posAbsolute := "Unit1.Em4.ControlNodes".cm.axisCommand.anodeMainPnP1AxisY.posAbsoluteSummary;
END_REGION

REGION Network 110: CmAnodeMainPnP2AxisY Interlock Summary
